(* CoDeSys 2.3.9.41 project: Projmodliv.pro *)
(* Libraries: STANDARD.LIB 4.10.05 10:14:46, IECSFC.LIB 13.4.06 14:51:28, SYSLIBTIME.LIB 12.2.21 12:34:31, SYSTASKINFO.LIB 20.2.06 12:31:38, ANALYZATION.LIB 5.10.99 08:05:06, SYSLIBCALLBACK.LIB 20.2.06 12:31:08, ComService.lib 12.2.21 12:39:42, SysLibCom.lib 12.2.21 12:35:47, ModBus.lib 12.2.21 12:36:21, Util.lib 18.5.10 14:14:28 *)

(* PLC configuration (modules and I/O channels)
DI1 AT %IB0.0 [ByteInput] 8 discrete inputs
Discrete output - relay [ID102] node 1, in %IB1 out %QB1 {PinCount = 1; SafeValueBool = FALSE; Visibility = No}
  DO1 AT %QX1.0 [BitOutput] relay
Discrete output - relay [ID102] node 2, in %IB2 out %QB2 {PinCount = 1; SafeValueBool = FALSE; Visibility = No}
  AT %QX2.0 [BitOutput] relay
Discrete output - relay [ID102] node 3, in %IB3 out %QB3 {PinCount = 1; SafeValueBool = FALSE; Visibility = No}
  AT %QX3.0 [BitOutput] relay
Discrete output - relay [ID102] node 4, in %IB4 out %QB4 {PinCount = 1; SafeValueBool = FALSE; Visibility = No}
  AT %QX4.0 [BitOutput] relay
Discrete output - relay [ID102] node 5, in %IB5 out %QB5 {PinCount = 1; SafeValueBool = FALSE; Visibility = No}
  AT %QX5.0 [BitOutput] relay
  DO6 AT %QX6.0 [BitOutput] relay
AT %QX7.0 [BitOutput] Special output
AT %IW8.0 [WordInput] Cycle time in 100 mks
AT %IW8.1 [WordInput] Time to backup power down, s
AT %ID8.2 [FloatInput] Temp inside PLC
AT %IX8.3 [BitInput] Power status
AT %IX8.4 [BitInput] CPU is overloaded, optimize your programm or increase PLC cycle
AT %IW8.5 [WordInput] Free processor resourse mks in 1 cycle
RS-232 [COM2_USART] node 0, in %IB9.0.0 out %QB9.0.0 {CommunicationSpeed = 9600; Parity = NO PARITY CHECK; BitLength = 8 bits; StopLength = One stop bit; InterfaceType = RS232; FrameOriented = RTU; Timeout = 0; Visibility = No}
ReSlave0 AT %QW9.1.0 [WordOutput]
ReSlave1 AT %QW9.2.0 [WordOutput]
ReSlave2 AT %QW9.3.0 [WordOutput]
ReSlave3 AT %QW9.4.0 [WordOutput]
ReSlave4 AT %QW9.5.0 [WordOutput]
ReSlave5 AT %QW9.6.0 [WordOutput]
ReSlave6 AT %QW9.7.0 [WordOutput]
ReSlave7 AT %QW9.8.0 [WordOutput]
ReSlave8 AT %QW9.9.0 [WordOutput]
ReSlave9 AT %QW9.10.0 [WordOutput]
ReSlave10 AT %QW9.11.0 [WordOutput]
ReSlave11 AT %QW9.12.0 [WordOutput]
ReSlave12 AT %QW9.13.0 [WordOutput]
ReSlave13 AT %QW9.14.0 [WordOutput]
ReSlave14 AT %QW9.15.0 [WordOutput]
ReSlave15 AT %QW9.16.0 [WordOutput]
ReSlave16 AT %QW9.17.0 [WordOutput]
ReSlave17 AT %QW9.18.0 [WordOutput]
ReSlave18 AT %QW9.19.0 [WordOutput]
ReSlave19 AT %QW9.20.0 [WordOutput]
ReSlave20 AT %QW9.21.0 [WordOutput]
ReSlave21 AT %QW9.22.0 [WordOutput]
ReSlave22 AT %QW9.23.0 [WordOutput]
ReSlave23 AT %QW9.24.0 [WordOutput]
ReSlave24 AT %QW9.25.0 [WordOutput]
ReSlave25 AT %QW9.26.0 [WordOutput]
ReSlave26 AT %QW9.27.0 [WordOutput]
ReSlave27 AT %QW9.28.0 [WordOutput]
ReSlave28 AT %QW9.29.0 [WordOutput]
ReSlave29 AT %QW9.30.0 [WordOutput]
ReSlave30 AT %QW9.31.0 [WordOutput]
ReSlave31 AT %QW9.32.0 [WordOutput]
ReSlave32 AT %QW9.33.0 [WordOutput]
ReSlave33 AT %QW9.34.0 [WordOutput]
*)

(* Global variable list: Global_Variables *)
VAR_GLOBAL

	port_opened:  BYTE := 0;
	Settings:COMSETTINGS;
      	com_num: PORTS:=0;
	COM_SERVICE1: COM_SERVICE;

	port_opened2:  BYTE := 0;
	Settings2:COMSETTINGS;
      	com_num2: PORTS:=1;
	COM_SERVICE2: COM_SERVICE;


	ModBusWriteMultiReg232: MB_WR_REGS;
	TonConnect232:ARRAY[0..10] OF  TON;
	ToffConnect232:ARRAY[0..10] OF  TOF;
	ConnectionStatus232:ARRAY[0..10] OF  BOOL;
	Buffer232: ARRAY[0..255] OF BYTE;
	Cmpl232: ARRAY[0..10] OF BOOL;
	Err232: ARRAY[0..10] OF BYTE;
       SCADAData:ARRAY[0..70] OF WORD;

	Buffer: ARRAY[0..255] OF BYTE;
	Cmpl: ARRAY[0..30] OF BOOL;
	Err: ARRAY[0..30] OF BYTE;
	i: BYTE;
	j: BYTE;

      TonConnect: ARRAY[0..3] OF TON;
	ToffConnect: ARRAY[0..3] OF TOF;
	ConnectionStatus: ARRAY [0..3] OF BOOL;



	ModBusWriteMultiCoil: ARRAY[0..1] OF MB_WR_COILS;
	ModBusReadHoldReg: ARRAY[0..10] OF MB_RD_HOLD_REGS;
	ModBusWriteMultiReg: ARRAY[0..10] OF MB_WR_REGS;
      NumberSend: BYTE;

	DisplayData:ARRAY[0..100] OF WORD;

       TimeOut: TIME := T#30ms;

       Out1: WORD;
	 In1: WORD;
       In2: WORD;
	PLCtime:ARRAY[0..10] OF WORD;

      BKDU_KTV:  ARRAY [0..1] OF WORD;  (*BKDU_KTV[0], 5*)

       LocalTime: CurTime;
	TimeL: SysTime64;

	CommCycleTime: SysTime64;
	CommCycleTimePrev: SysTime64;

       ServisWork: BOOL;

	Stop: BOOL;
	StopTime: TIME:=T#1S;
	Zashtibovka: BOOL;
	Zash: BOOL;
	ZashTime: TIME := T#10S;
	KTB: BOOL;
	KTBTime: TIME := T#1S;
	DKS: BOOL;
	DKSTime: TIME := T#10S;
	BOP: INT;
	SirVPN: BOOL;
       AvSirVPN: BOOL;
	TK1: INT;
	TK2: INT;
	TK3: INT;
	TK4: INT;
	KTBStopAv: BOOL;
	KTBStopAvKZ: BOOL;
	KTBCurrent: UINT;
	KTBPower: UINT;
       StopSignal: TP;

	KTBRabotaet: BOOL;
	RazgonStop: BOOL;
	RabotaSpeedStop: BOOL;
	PuskKonveera: BOOL;
	KSLsrabotal: BOOL;
	KSLKZ: BOOL;
	PodtvPusk4: BOOL;
	PodtvPusk3: BOOL;
	myTP22: BOOL;
	PodtvPusk1: BOOL;
	PodtvPusk2: BOOL;
	PP1: BOOL;
	PP2: BOOL;
	PP3: BOOL;
	PP4: BOOL;
	SbrosRazgona: BOOL;
	Parol: UINT := 0;
	ParolStep: UINT := 0;
	Parol1: UINT := 0;
	Parol2: UINT := 0;
	Parol3: UINT := 0;
	GlobalAvariaStop: BOOL;
	DistSignal: BOOL;
	P1Signal: BOOL;

       myTP100: TON;




END_VAR

VAR_GLOBAL RETAIN

	GetTime: CurTimeEx;
	TimeAndDate: SystemTimeDate;
	Sys_Time: SysTime64;
	set_time: BOOL;
	set_date: BOOL;
	MM: UINT:=10;
	SS: UINT;
	HH: UINT:=10;
	D: UINT:=10;
	M: UINT:=10;
	YY: UINT:=20;







	xDO6: TIME := T#6s;
	ZashtibovkaTime: TIME := T#5S;
	RazgonTime: TIME:=T#5s;
	AvariaTime: TIME:=T#10s;
	PuskTime: TIME := T#5s;
	KTBSht: UINT := 5;
	TipK1: UINT := 0;
       TipK1P: TIME:=T#0.2s;
	TipK1T: UINT := 0;
       TipK1UP: TIME:=T#1s;
	TipK2: UINT := 0;
       TipK2P: TIME:=T#0.2s;
	TipK2T: UINT := 0;
       TipK2UP: TIME:=T#1s;
       TipK3: UINT := 0;
       TipK3P: TIME:=T#0.2s;
	TipK3T: UINT := 0;
       TipK3UP: TIME:=T#1s;
       TipK4: UINT := 0;
       TipK4P: TIME:=T#0.2s;
	TipK4T: UINT := 0;
       TipK4UP: TIME:=T#1s;
	NomSpeed: UINT := 20;
	TipDat: UINT:=1;
	DiamKDKS: UINT:=123;
	ImpDKS: UINT:=30;
       Rez: UINT:=300;

	xDO6q: TIME := T#6s;
	ZashtibovkaTimeq: TIME := T#5S;
	RazgonTimeq: TIME:=T#5s;
	AvariaTimeq: TIME:=T#10s;
	PuskTimeq: TIME := T#5s;
	KTBShtq: UINT := 5;
	TipK1q: UINT := 0;
	TipK1Pq: TIME:=T#0.2s;
	TipK1Tq: UINT := 0;
       TipK1UPq: TIME:=T#1s;
	TipK2q: UINT := 0;
       TipK2Pq: TIME:=T#0.2s;
	TipK2Tq: UINT := 0;
       TipK2UPq: TIME:=T#1s;
       TipK3q: UINT := 0;
       TipK3Pq: TIME:=T#0.2s;
	TipK3Tq: UINT := 0;
       TipK3UPq: TIME:=T#1s;
       TipK4q: UINT := 0;
       TipK4Pq: TIME:=T#0.2s;
	TipK4Tq: UINT := 0;
       TipK4UPq: TIME:=T#1s;
	NomSpeedq: UINT := 20;
	TipDatq: UINT:=1;
	DiamKDKSq: UINT:=123;
	ImpDKSq: UINT:=30;
       Rezq: UINT:=300;

	xDO6qi: UINT :=60;
	ZashtibovkaTimeqi: UINT := 50;
	RazgonTimeqi: UINT:=50;
	AvariaTimeqi: WORD:=10;
	PuskTimeqi: WORD := 50;
      TipK1Pqi: UINT:=2;
      TipK1UPqi: UINT:=10;
      TipK2Pqi: UINT:=2;
      TipK2UPqi: UINT:=10;
      TipK3Pqi: UINT:=2;
      TipK3UPqi: UINT:=10;
      TipK4Pqi: UINT:=2;
      TipK4UPqi: UINT:=10;


      Reztek:UINT:=300;

	xDO6Po: UINT :=60;
	ZashtibovkaTimePo: UINT := 50;
	RazgonTimePo: UINT:=50;
	AvariaTimePo: WORD:=10;
	PuskTimePo: WORD := 50;
      TipK1PPo: UINT:=2;
      TipK1UPPo: UINT:=10;
      TipK2PPo: UINT:=2;
      TipK2UPPo: UINT:=10;
      TipK3PPo: UINT:=2;
      TipK3UPPo: UINT:=10;
      TipK4PPo: UINT:=2;
      TipK4UPPo: UINT:=10;


	KTB0: UINT;

        Smoke_sensorQ: BOOL:=TRUE;
       Methane_sensorQ:BOOL:=TRUE;
       Guard_sensorQ:BOOL:=TRUE;
       Add_avarQ:BOOL:=TRUE;



       Smoke_sensor: BOOL:=TRUE;
       Methane_sensor:BOOL:=TRUE;
       Guard_sensor:BOOL:=TRUE;
       Add_avar:BOOL:=TRUE;

END_VAR

(* POU PLC_PRG, ST *)
PROGRAM PLC_PRG
VAR
	myTON:TON;
	myR_TRIG:R_TRIG;
	FI1: INT:=0;

	start: BOOL;

	x: UINT;
	external_event: BOOL;

	ProverkaPuska: INT;
	AvariaSbros: INT;
	AvariaBOP: BOOL;
	ForwardSignal: Signal;
	StartForwardSignal: BOOL;
	Dsignal: BOOL;

       WorkModeF: F_TRIG;
	WorkModeT: R_TRIG;
	StopDist: BOOL;
	RabotaDist: BOOL;
	AvariaDist: BOOL;
	PuskKonveeraN: BOOL;
	a: INT;
	RezNastr: BOOL;
	SwitchWorkMode: BOOL;
	TpAvaria: TP;
	AvariaSirena: BOOL;
      TPBOP: TON;
      TRIGBOP: R_TRIG;
       StopTRIG: F_TRIG;
       StopTRIGr: R_TRIG;
       DistTrig1: R_TRIG;
       DistTrig2: R_TRIG;
	Metka: INT;
      Servis : TON;
      Servis2: TON;
      Servis1: R_TRIG;
	bcdT: INT;
	qwerty: BOOL;
	qwertyTP: TON;
	SmokeAv: BOOL;
	MethanAv: BOOL;
	GuardAv: BOOL;
	AddAv: BOOL;
       StopDistTrig: R_TRIG;
END_VAR
LocalTime(SystemTime:=TimeL );							(*	Функция времени	*)
IF start=0 THEN
	Init();						(*	Открытие порта RS-485	*)
	start:=1;
END_IF
Link();


DisplayData[51].13:=TRUE;

DisplayData[51].6:=TRUE;
DisplayData[51].2:=(ConnectionStatus[0]);       (*БВВ*)
DisplayData[51].3:=(ConnectionStatus[1]);       (*БКДУ*)
DisplayData[51].4:=(ConnectionStatus[2]);       (*ЗАШТЫБОВКА*)
(*IF pollCheclPLZ =16#00FE THEN
pollCheclPLZ :=16#00FF;
ELSE	
pollCheclPLZ :=16#00FE;
END_IF*)
IF DisplayData[23].5=FALSE AND In1.0=TRUE THEN
Servis(In:=In1.4, PT:=t#3s);
IF Servis.Q AND In1.4 THEN
Servis2(In:=In1.1, PT:=t#6s);
Servis1(CLK:=Servis2.Q);
IF Servis1.Q AND In1.4 THEN
ServisWork:=TRUE;
AvariaSbros:=0;

IF TipK1<>2 THEN
Out1.0:=TRUE;
END_IF

IF TipK2<>2 THEN
Out1.1:=TRUE;
END_IF

IF TipK3<>2 THEN
Out1.2:=TRUE;
END_IF

IF TipK4<>2 THEN
Out1.3:=TRUE;
END_IF
END_IF
ELSIF DisplayData[23].5=TRUE AND In1.0=FALSE THEN
ServisWork:=FALSE;
END_IF
END_IF

IF  ServisWork=FALSE THEN
DisplayData[51].5:=FALSE;
ELSE
DisplayData[51].5:=TRUE;
END_IF


StopTRIG(CLK:=In1.0);
StopTRIGr(CLK:=DisplayData[23].5=FALSE);
IF StopTRIGr.Q (*AND StopSignal.Q =FALSE*) THEN
Stop:=FALSE;
END_IF

IF DO1=TRUE THEN
DisplayData[24].15:=TRUE;
ELSIF DO1=FALSE THEN
DisplayData[24].15:=FALSE;
END_IF

IF in1.0=FALSE THEN
DisplayData[23].5:=FALSE;
END_IF

IF ((In1.0=FALSE OR StopTRIG.Q) OR ((KTBRabotaet=FALSE) AND AvariaSbros<>1))  AND ServisWork=FALSE  (*OR StopDist=TRUE*) (*OR RazgonStop=TRUE OR RabotaSpeedStop=TRUE OR KTBRabotaet=FALSE  OR KSLsrabotal=TRUE *)(* OR ((KTBRabotaet=FALSE OR (KSLsrabotal=TRUE AND KSLKZ=FALSE)) AND AvariaSbros<>1)*) THEN
StopDist:=FALSE;
PuskKonveera:=FALSE;
Stop:=TRUE;
sirVPN:=FALSE;
	DO1:=FALSE;
	Out1.0:=FALSE;
	Out1.1:=FALSE;
	Out1.2:=FALSE;
	Out1.3:=FALSE;
RazgonStop:=FALSE;
RabotaSpeedStop:=FALSE;
FI1:=0;
AvariaSbros:=0;

PuskKonveera:=FALSE;

AvariaBOP:=FALSE;

AvariaDist:=FALSE;
P1Signal:=FALSE;

PP1:=TRUE;
PP2:=TRUE;
PP3:=TRUE;
PP4:=TRUE;

Zash:=FALSE;

(*DisplayData[23].5:=TRUE;*)

SbrosRazgona:=TRUE;

PuskKonveera:=FALSE;

GlobalAvariaStop:=FALSE;
SwitchWorkMode:=FALSE;
AvariaSirena:=FALSE;


myTP100(In:=FALSE);
(*IF KTBRabotaet=FALSE  OR KSLsrabotal=TRUE THEN
DisplayData[23].2 :=TRUE;
END_IF
IF RazgonStop=TRUE THEN
END_IF
IF RabotaSpeedStop=TRUE THEN
END_IF*)
ELSIF (RazgonStop=TRUE OR RabotaSpeedStop=TRUE OR KTBstopAvKZ=TRUE OR AvariaBOP=TRUE
(*OR PodtvPusk1=FALSE OR PodtvPusk2=FALSE OR Po           dtvPusk3=FALSE OR PodtvPusk4=FALSE*)
OR  PP1=FALSE OR PP2=FALSE OR PP3=FALSE OR PP4=FALSE OR AvariaDist=TRUE
OR RezNastr=TRUE OR SwitchWorkMode=TRUE
 OR  ConnectionStatus[0]=TRUE OR  ConnectionStatus[1]=TRUE OR ConnectionStatus[2]=TRUE OR SmokeAv=TRUE OR MethanAv=TRUE
OR GuardAv=TRUE OR AddAv=TRUE  )
 AND ServisWork=FALSE THEN
GlobalAvariaStop:=TRUE;
PuskKonveera:=FALSE;
DO1:=FALSE;
Out1.0:=FALSE;
Out1.1:=FALSE;
Out1.2:=FALSE;
Out1.3:=FALSE;
FI1:=2;
AvariaSbros:=1;
DisplayData[23].5:=FALSE;
SbrosRazgona:=TRUE;
AvariaDist:=TRUE;
AvariaSirena:=TRUE;

(*ELSIF KTBRabotaet=FALSE  THEN
PuskKonveera:=FALSE;
DO1:=FALSE;
Out1.0:=FALSE;
Out1.1:=FALSE;
Out1.2:=FALSE;
Out1.3:=FALSE;
FI1:=0;
KTB:=TRUE;
ELSIF DI1.0=TRUE  AND DI1.0=FALSE THEN
PuskKonveera:=FALSE;
DO1:=FALSE;
Out1.0:=FALSE;
Out1.1:=FALSE;
Out1.2:=FALSE;
Out1.3:=FALSE;
FI1:=0;
DKS:=TRUE;*)
ELSIF (SmokeAv=FALSE AND MethanAv=FALSE
AND GuardAv=FALSE AND AddAv=FALSE  )
 AND ServisWork=FALSE AND in1.5=TRUE AND KSLsrabotal=TRUE THEN
DisplayData[23].5:=FALSE;
PuskKonveera:=FALSE;
DO1:=FALSE;
Out1.0:=FALSE;
Out1.1:=FALSE;
Out1.2:=FALSE;
Out1.3:=FALSE;
P1Signal:=FALSE;
SbrosRazgona:=TRUE;
Stop:=TRUE;
AvariaSirena:=TRUE;
myTP100(In:=FALSE);
RazgonStop:=FALSE;
RabotaSpeedStop:=FALSE;
FI1:=0;

ELSIF (SmokeAv=FALSE AND MethanAv=FALSE
AND GuardAv=FALSE AND AddAv=FALSE  )
 AND ServisWork=FALSE AND in1.5=TRUE AND Zash=TRUE THEN
DisplayData[23].5:=FALSE;
PuskKonveera:=FALSE;
DO1:=FALSE;
Out1.0:=FALSE;
Out1.1:=FALSE;
Out1.2:=FALSE;
Out1.3:=FALSE;
P1Signal:=FALSE;
SbrosRazgona:=TRUE;
Stop:=TRUE;
AvariaSirena:=TRUE;
myTP100(In:=FALSE);
RazgonStop:=FALSE;
RabotaSpeedStop:=FALSE;
FI1:=0;

ELSIF (SmokeAv=FALSE AND MethanAv=FALSE
AND GuardAv=FALSE AND AddAv=FALSE  )
 AND ServisWork=FALSE AND in1.5=TRUE AND KSLKZ=TRUE THEN
DisplayData[23].5:=FALSE;
PuskKonveera:=FALSE;
DO1:=FALSE;
Out1.0:=FALSE;
Out1.1:=FALSE;
Out1.2:=FALSE;
Out1.3:=FALSE;
P1Signal:=FALSE;
SbrosRazgona:=TRUE;
Stop:=TRUE;
AvariaSirena:=TRUE;
myTP100(In:=FALSE);
RazgonStop:=FALSE;
RabotaSpeedStop:=FALSE;
FI1:=0;

ELSIF In1.0=FALSE OR In1.4=FALSE AND ServisWork=TRUE THEN
ServisWork:=FALSE;
ELSE
DisplayData[23].5:=TRUE;
AvariaSirena:=FALSE;
(*ELSIF (KTBRabotaet=FALSE OR (KSLsrabotal=TRUE AND KSLKZ=FALSE)) AND AvariaSbros<>1  THEN
PuskKonveera:=FALSE;
Stop:=TRUE;
DO1:=FALSE;
Out1.0:=FALSE;
Out1.1:=FALSE;
Out1.2:=FALSE;
Out1.3:=FALSE;*)
END_IF

IF In1.3=TRUE (*AND ServisWork=FALSE*) THEN
RezNastr:=FALSE;

IF Zashtibovka THEN
DisplayData[23].4:=FALSE;
ELSE
DisplayData[23].4:=TRUE;
END_IF

IF KTBRabotaet=FALSE OR KSLsrabotal=TRUE OR KSLKZ=TRUE OR KTBStopAvKZ THEN
DisplayData[23].2 :=FALSE;
ELSE
DisplayData[23].2 :=TRUE;
END_IF

IF RazgonStop=TRUE OR RabotaSpeedStop=TRUE THEN
DisplayData[23].3:=FALSE;
ELSE
DisplayData[23].3:=TRUE;
END_IF

(*DisplayData[23].3:=DI1.0;*)
(*IF (Zash=FALSE OR KTBRabotaet=TRUE OR RazgonStop=FALSE OR RabotaSpeedStop=FALSE OR KSLsrabotal=FALSE) AND AvariaSbros=0 THEN
DisplayData[23].5:=TRUE;
ELSE
DisplayData[23].5:=FALSE;
END_IF*)


IF In1.4=TRUE THEN
SirVPN:=TRUE;
ELSIF In1.4=FALSE THEN
SirVPN:=FALSE;
END_IF

(*IF In1.0=FALSE THEN
SirVPN:=FALSE;
AvariaSirena:=FALSE;
DO6:=FALSE;
AvSirVPN:=FALSE;
END_IF *)
IF In1.2=FALSE THEN
DisplayData[24].4:=TRUE;
DisplayData[24].5:=FALSE;

(*IF FI1=2 THEN
Stop:=TRUE;
DO1:=FALSE;
Out1.0:=FALSE;
Out1.1:=FALSE;
Out1.2:=FALSE;
Out1.3:=FALSE;
END_IF*)


IF In1.1=TRUE AND FI1=0 AND In1.2=FALSE (*AND DI1.0=FALSE*) AND KSLsrabotal=FALSE (*AND KTBRabotaet=FALSE*) AND KTBstopAvKZ=FALSE  AND Zash=FALSE AND In1.0=TRUE AND AvariaSbros=0 THEN
PuskKonveera:=TRUE;
(*DO1:=TRUE;*)
Stop:=FALSE;
FI1:=1;
SbrosRazgona:=FALSE;
ELSIF In1.1=FALSE AND FI1=1  AND In1.2=FALSE (*AND DI1.0=FALSE*) AND  KSLsrabotal=FALSE (*AND KTBRabotaet=FALSE*) AND KTBstopAvKZ=FALSE AND Zash=FALSE AND In1.0=TRUE AND AvariaSbros=0 THEN
PuskKonveera:=TRUE;
(*DO1:=TRUE;*)
Stop:=FALSE;
SbrosRazgona:=FALSE;
ELSIF In1.1=TRUE AND FI1=1 AND In1.2=FALSE (*AND DI1.0=FALSE*) AND KSLsrabotal=FALSE (*AND KTBRabotaet=FALSE*) AND KTBstopAvKZ=FALSE  AND Zash=FALSE AND In1.0=TRUE AND AvariaSbros=0 THEN
PuskKonveera:=TRUE;
(*DO1:=TRUE;*)
Stop:=FALSE;
SbrosRazgona:=FALSE;
END_IF



ELSIF In1.2=TRUE THEN
DisplayData[24].4:=FALSE;
DisplayData[24].5:=TRUE;
TPBOP(IN:=DI1.1=TRUE AND DI1.2=TRUE , PT:=t#1.0s);
TRIGBOP(CLK:=TPBOP.Q);
DistTrig1(CLK:=(DI1.1=TRUE AND DI1.2=FALSE));
DistTrig2(CLK:=(DI1.1=FALSE AND DI1.2=TRUE));
(*IF FI1=1 THEN
DO1:=FALSE;
Out1.0:=FALSE;
Out1.1:=FALSE;
Out1.2:=FALSE;
Out1.3:=FALSE;
Stop:=TRUE;
END_IF*)
IF DI1.1=TRUE AND DI1.2=FALSE THEN
DisplayData[24].1:=FALSE;
DisplayData[24].2:=TRUE;
DisplayData[24].3:=FALSE;
DisplayData[23].1:=FALSE;
DisplayData[24].6:=FALSE;
ELSIF DI1.1=FALSE AND DI1.2=TRUE THEN
DisplayData[24].1:=TRUE;
DisplayData[24].2:=FALSE;
DisplayData[24].3:=FALSE;
DisplayData[23].1:=FALSE;
DisplayData[24].6:=FALSE;
ELSIF DI1.1=TRUE AND DI1.2=TRUE THEN

DisplayData[24].1:=FALSE;
DisplayData[24].2:=FALSE;
DisplayData[24].3:=FALSE;
DisplayData[24].6:=TRUE;
DisplayData[23].1:=FALSE;
ELSIF DI1.1=FALSE AND DI1.2=FALSE THEN

DisplayData[23].1:=TRUE;
DisplayData[24].1:=FALSE;
DisplayData[24].2:=FALSE;
DisplayData[24].3:=TRUE;
DisplayData[24].6:=FALSE;
END_IF

IF DI1.1=TRUE AND DI1.2=FALSE AND DistTrig1.Q  AND AvariaSbros=0 AND In1.0=TRUE (*AND PuskKonveera=FALSE*) AND AvariaDist=FALSE (*AND Metka=0*) THEN
(*PuskKonveera:=TRUE;*)
(*DO1:=TRUE;*)
(*FI1:=2;*)
RabotaDist:=TRUE;
(*DisplayData[24].1:=FALSE;
DisplayData[24].2:=TRUE;
DisplayData[24].3:=FALSE;
DisplayData[23].1:=FALSE;
DisplayData[24].6:=FALSE;*)
(* Metka:=2;*)
ELSIF DI1.1=FALSE AND DI1.2=TRUE AND DistTrig2.Q AND AvariaSbros=0 AND In1.0=TRUE (*AND PuskKonveera=TRUE  AND RabotaDist=FALSE*) AND AvariaDist=FALSE(* AND Metka=1*) THEN
PuskKonveera:=TRUE;
(*DO1:=TRUE;*)
(*FI1:=2;*)
RabotaDist:=FALSE;
(*DisplayData[24].1:=TRUE;
DisplayData[24].2:=FALSE;
DisplayData[24].3:=FALSE;
DisplayData[23].1:=FALSE;
DisplayData[24].6:=FALSE;*)
SbrosRazgona:=FALSE;
(*Metka:=1;*)

(*PuskKonveera:=TRUE;*)
(*DO1:=TRUE;
FI1:=2;*)


ELSIF (TRIGBOP.Q AND In1.0=TRUE AND AvariaDist=FALSE) OR StopTRIG.Q THEN

Metka:=0;
ProverkaPuska:=0;
(*DisplayData[23].1:=FALSE;*)
DO1:=FALSE;
Out1.0:=FALSE;
Out1.1:=FALSE;
Out1.2:=FALSE;
Out1.3:=FALSE;
(*DisplayData[24].1:=FALSE;
DisplayData[24].2:=FALSE;
DisplayData[24].3:=FALSE;
DisplayData[24].6:=TRUE;*)
StopDist:=TRUE;

SbrosRazgona:=TRUE;
PuskKonveera:=FALSE;
DisplayData[63].13:=TRIGBOP.Q;

(*END_IF*)
ELSIF DI1.1=FALSE AND DI1.2=FALSE AND In1.0=TRUE THEN
DO1:=FALSE;
Out1.0:=FALSE;
Out1.1:=FALSE;
Out1.2:=FALSE;
Out1.3:=FALSE;
AvariaBOP:=TRUE;
(*BOP:=1;
FI1:=1;*)
(*DisplayData[23].1:=TRUE;
DisplayData[24].1:=FALSE;
DisplayData[24].2:=FALSE;
DisplayData[24].3:=TRUE;
DisplayData[24].6:=FALSE;*)
END_IF
END_IF

IF In2<=Reztek THEN
Zashtibovka:=TRUE;
(*B392:=TRUE;*)
ELSIF In2>Reztek THEN
Zashtibovka:=FALSE;
(*B392:=FALSE;*)
END_IF

ELSIF In1.3=FALSE THEN

DO1:=FALSE;
Out1.0:=FALSE;
Out1.1:=FALSE;
Out1.2:=FALSE;
Out1.3:=FALSE;
SirVPN:=FALSE;
RezNastr:=TRUE;
END_IF

IF In1.6=TRUE (*AND TipK1T<>1*) THEN
DisplayData[23].9:=TRUE;
DisplayData[23].10:=FALSE;
ELSIF In1.6=FALSE (*AND TipK1T<>1*) THEN
DisplayData[23].9:=FALSE;
DisplayData[23].10:=TRUE;
END_IF
IF In1.7=TRUE (*AND TipK2T <>1*) THEN
DisplayData[23].11:=TRUE;
DisplayData[23].12:=FALSE;
ELSIF In1.7=FALSE (*AND TipK2T<>1*) THEN
DisplayData[23].11:=FALSE;
DisplayData[23].12:=TRUE;
END_IF
IF In1.8=TRUE (*AND TipK3T<>1*) THEN
DisplayData[23].13:=TRUE;
DisplayData[23].14:=FALSE;
ELSIF In1.8=FALSE (*AND TipK3T<>1*) THEN
DisplayData[23].13:=FALSE;
DisplayData[23].14:=TRUE;
END_IF
IF In1.9=TRUE (*AND TipK4T<>1*) THEN
DisplayData[23].15:=TRUE;
DisplayData[24].0:=FALSE;
ELSIF In1.9=FALSE (*AND TipK4T<>1*) THEN
DisplayData[23].15:=FALSE;
DisplayData[24].0:=TRUE;
END_IF
(********************************************************************************************************
IF TipK1=1 AND DO6=TRUE THEN
out1.0:=TRUE;
ELSIF TipK1<>1 AND DO6=FALSE THEN
out1.0:=FALSE;
END_IF

IF TipK2=1 AND DO6=TRUE THEN
out1.1:=TRUE;
ELSIF TipK2<>1  AND DO6=FALSE THEN
out1.1:=FALSE;
END_IF

IF TipK3=1 AND DO6=TRUE THEN
out1.2:=TRUE;
ELSIF TipK3<>1 AND DO6=FALSE THEN
out1.2:=FALSE;
END_IF

IF TipK4=1 AND DO6=TRUE THEN
out1.3:=TRUE;
ELSIF TipK4<>1 AND DO6=FALSE THEN
out1.3:=FALSE;
END_IF
 ***********************************************************************************************************************)
IF out1.0=TRUE THEN
DisplayData[24].10:=TRUE;
ELSIF out1.0=FALSE THEN
DisplayData[24].10:=FALSE;
END_IF

IF out1.1=TRUE THEN
DisplayData[24].11:=TRUE;
ELSIF out1.1=FALSE THEN
DisplayData[24].11:=FALSE;
END_IF
IF out1.2=TRUE THEN
DisplayData[24].12:=TRUE;
ELSIF out1.2=FALSE THEN
DisplayData[24].12:=FALSE;
END_IF

IF out1.3=TRUE THEN
DisplayData[24].13:=TRUE;
ELSIF out1.3=FALSE THEN
DisplayData[24].13:=FALSE;
END_IF


IF DO6=TRUE THEN
(*Sirena1:='ВКЛ';*)
DisplayData[23].7:=TRUE;
DisplayData[23].8:=FALSE;
ELSIF DO6=FALSE THEN
(*Sirena1:='ВЫКЛ';*)
DisplayData[23].7:=FALSE;
DisplayData[23].8:=TRUE;
END_IF



(**)
IF Smoke_sensor THEN
IF in1.10 THEN
DisplayData[66].8:=TRUE;
DisplayData[66].9:=FALSE;
ELSE
DisplayData[66].8:=FALSE;
DisplayData[66].9:=TRUE;
END_IF
ELSE
IF in1.10=FALSE THEN
DisplayData[66].8:=TRUE;
DisplayData[66].9:=FALSE;
ELSE
DisplayData[66].8:=FALSE;
DisplayData[66].9:=TRUE;
END_IF
END_IF

IF Methane_sensor THEN
IF in1.14 THEN
DisplayData[66].10:=TRUE;
DisplayData[66].11:=FALSE;
ELSE
DisplayData[66].10:=FALSE;
DisplayData[66].11:=TRUE;
END_IF
ELSE
IF in1.14=FALSE THEN
DisplayData[66].10:=TRUE;
DisplayData[66].11:=FALSE;
ELSE
DisplayData[66].10:=FALSE;
DisplayData[66].11:=TRUE;
END_IF
END_IF

IF Guard_sensor THEN
IF in1.15 THEN
DisplayData[66].12:=TRUE;
DisplayData[66].13:=FALSE;
ELSE
DisplayData[66].12:=FALSE;
DisplayData[66].13:=TRUE;
END_IF
ELSE
IF in1.15=FALSE THEN
DisplayData[66].12:=TRUE;
DisplayData[66].13:=FALSE;
ELSE
DisplayData[66].12:=FALSE;
DisplayData[66].13:=TRUE;
END_IF
END_IF

IF  Add_avar THEN
IF in1.5 THEN
DisplayData[66].14:=TRUE;
DisplayData[66].15:=FALSE;
ELSE
DisplayData[66].14:=FALSE;
DisplayData[66].15:=TRUE;
END_IF
ELSE
IF in1.15=FALSE THEN
DisplayData[66].14:=TRUE;
DisplayData[66].15:=FALSE;
ELSE
DisplayData[66].14:=FALSE;
DisplayData[66].15:=TRUE;
END_IF
END_IF

IF DisplayData[66].9=TRUE THEN
SmokeAv:=TRUE;
DisplayData[67].0:=TRUE;
DisplayData[67].1:=FALSE;
ELSE
SmokeAv:=FALSE;
DisplayData[67].0:=FALSE;
DisplayData[67].1:=TRUE;
END_IF

IF DisplayData[66].11=TRUE THEN
MethanAv:=TRUE;
DisplayData[67].2:=TRUE;
DisplayData[67].3:=FALSE;
ELSE
MethanAv:=FALSE;
DisplayData[67].2:=FALSE;
DisplayData[67].3:=TRUE;
END_IF

IF DisplayData[66].13=TRUE THEN
GuardAv:=TRUE;
DisplayData[67].4:=TRUE;
DisplayData[67].5:=FALSE;
ELSE
GuardAv:=FALSE;
DisplayData[67].4:=FALSE;
DisplayData[67].5:=TRUE;
END_IF

IF DisplayData[66].15=TRUE THEN
AddAv:=TRUE;
DisplayData[67].6:=TRUE;
DisplayData[67].7:=FALSE;
ELSE
AddAv:=FALSE;
DisplayData[67].6:=FALSE;
DisplayData[67].7:=TRUE;
END_IF
(**)

Schet();
Timers();
Impuls();
KTBlog();
PuskLogick();
SlaveRS232();


(*IF TK1=1 THEN
IF ProverkaPuska=1 THEN
END_IF
END_IF*)

(*ForwardSignal(Enable:=StartForwardSignal ,Quantity:=4 ,TimeLow:=T#500ms ,TimeHigh:=T#500ms , TimeHighLast:=T#500ms ,Out=> );
Dsignal:=ForwardSignal.Out;
*)
(*
WorkModeT*) 
WorkModeT(CLK:=In1.2);
IF WorkModeT.Q THEN
SwitchWorkMode:=TRUE;
DisplayData[24].1:=FALSE;
DisplayData[24].2:=FALSE;
DisplayData[24].3:=FALSE;
DisplayData[24].6:=TRUE;
DisplayData[51].1:=TRUE;
END_IF

WorkModeF(CLK:=In1.2);
IF WorkModeF.Q THEN
SwitchWorkMode:=TRUE;
DisplayData[24].1:=FALSE;
DisplayData[24].2:=FALSE;
DisplayData[24].3:=FALSE;
DisplayData[24].6:=FALSE;
DisplayData[51].1:=FALSE;
END_IF

IF DI1.3 AND In1.2 THEN
DistSignal:=TRUE;
ELSIF (DI1.3=FALSE AND In1.2) OR (DI1.3 AND In1.2=FALSE) THEN
DistSignal:=FALSE;
END_IF





TpAvaria(IN:=AvariaSirena , PT:=AvariaTime);
IF TpAvaria.Q THEN

IF RazgonStop=TRUE OR RabotaSpeedStop=TRUE THEN
ForwardSignal(Enable:=TpAvaria.Q ,Quantity:=4 ,TimeLow:=T#500ms ,TimeHigh:=T#500ms , TimeHighLast:=T#500ms ,Out=> );
AvSirVPN:=ForwardSignal.Out;
END_IF
IF Zash=TRUE THEN
ForwardSignal(Enable:=TpAvaria.Q ,Quantity:=3 ,TimeLow:=T#500ms ,TimeHigh:=T#500ms , TimeHighLast:=T#500ms ,Out=> );
AvSirVPN:=ForwardSignal.Out;
END_IF
IF KTBstopAvKZ=TRUE OR KSLKZ=TRUE OR KSLsrabotal OR  SmokeAv=TRUE OR MethanAv=TRUE OR GuardAv=TRUE OR AddAv=TRUE THEN (**)
(*ForwardSignal(Enable:=TpAvaria.Q ,Quantity:=3 ,TimeLow:=T#500ms ,TimeHigh:=T#500ms , TimeHighLast:=T#500ms ,Out=> );*)
AvSirVPN:=TpAvaria.Q;
END_IF
IF AvariaBOP=TRUE THEN
ForwardSignal(Enable:=TpAvaria.Q ,Quantity:=3 ,TimeLow:=T#500ms ,TimeHigh:=T#500ms , TimeHighLast:=T#500ms ,Out=> );
AvSirVPN:=ForwardSignal.Out;
END_IF
IF  PP1=FALSE OR PP2=FALSE OR PP3=FALSE OR PP4=FALSE THEN (**)
(*ForwardSignal(Enable:=TpAvaria.Q ,Quantity:=3 ,TimeLow:=T#500ms ,TimeHigh:=T#500ms , TimeHighLast:=T#500ms ,Out=> );*)
AvSirVPN:=TpAvaria.Q;
END_IF
(*ELSIF TpAvaria.Q=FALSE AND AvariaSbros=0 AND SirVPN=FALSE THEN
DO6:=SirVPN;*)
ELSE
AvSirVPN:=FALSE;
END_IF

DisplayData[64]:=In2;


DisplayData[62].10:=Zash;
DisplayData[62].11:=RazgonStop;
DisplayData[62].12:=RabotaSpeedStop;
DisplayData[62].13:=KTBstopAvKZ;
DisplayData[62].14:=KSLKZ;
DisplayData[62].15:=AvariaBOP;
DisplayData[63].0:=NOT PP1;
DisplayData[63].1:=NOT PP2;
DisplayData[63].2:=NOT PP3;
DisplayData[63].3:=NOT PP4;
DisplayData[63].4:=ConnectionStatus[0];
DisplayData[63].5:=ConnectionStatus[1];
DisplayData[63].6:=ConnectionStatus[2];
DisplayData[63].7:=KSLsrabotal;
DisplayData[63].9:=SmokeAv;
DisplayData[63].10:=MethanAv;
DisplayData[63].11:=GuardAv;
DisplayData[63].12:=AddAv;
END_PROGRAM

(* POU Signal, ST *)
FUNCTION_BLOCK Signal
VAR_INPUT
	Enable: BOOL;
	Quantity:BYTE;
	TimeLow: TIME;
	TimeHigh: TIME;
	TimeHighLast: TIME;
	Beep: BOOL;
END_VAR
VAR_OUTPUT
	Out: BOOL;
END_VAR
VAR
	TimeHihgInternal: TIME;
	Work: BOOL;
	Beepp:BLINK;
	BeepLatchQaun: BOOL;
	BeepQaun: BYTE;
END_VAR
IF (Enable OR  Beep)THEN
	Work:=TRUE;
	IF NOT(Beep) THEN
		Beep:=1;
	END_IF
	IF NOT(Out) THEN
		IF BeepLatchQaun THEN
			BeepLatchQaun:=0;
			BeepQaun:=BeepQaun+1;
		END_IF
	ELSE
		BeepLatchQaun:=1;
	END_IF
	IF BeepQaun=(Quantity-1) THEN
		TimeHihgInternal:=TimeHighLast;
	ELSE
		TimeHihgInternal:=TimeHigh;
	END_IF
	IF BeepQaun=Quantity THEN
		Work:=FALSE;
		Beep:=0;
		BeepQaun:=0;
	END_IF
	Beepp(ENABLE:=Beep, TIMELOW:=TimeLow , TIMEHIGH:=TimeHihgInternal, OUT=>Out );
ELSE
	Work:=FALSE;
	Beep:=0;
	BeepQaun:=0;
	Out:=0;
END_IF
END_FUNCTION_BLOCK

(* POU Init, ST *)
FUNCTION Init : BOOL
VAR_INPUT
END_VAR
VAR
END_VAR
WHILE port_opened=0 DO
	IF port_opened=0 THEN
		Settings.Port:=com_num;
		Settings.dwBaudRate:=57600;
		Settings.byParity:=0;
		Settings.dwTimeout:=0;
		Settings.byStopBits:=0;
		Settings.dwBufferSize:=0;
		Settings.dwScan:=0;
	END_IF
	COM_SERVICE1(Enable:=(port_opened=0) , Settings:=Settings , Task:=OPEN_TSK  );
	IF COM_SERVICE1.ready THEN
		port_opened:=2;
	END_IF
END_WHILE
END_FUNCTION

(* POU Link, ST *)
FUNCTION Link : BOOL
VAR_INPUT
END_VAR
VAR
	z: BYTE;
	a: BOOL;

END_VAR
CASE NumberSend OF
0:
	FOR z:=0 TO 70  BY 1 DO
		Buffer[z*2+1]:=WORD_TO_BYTE(DisplayData[z] AND 16#00FF);
		Buffer[z*2]:=WORD_TO_BYTE(SHR(DisplayData[z], 8));
	END_FOR
	ModBusWriteMultiReg[0](
		Enable:=TRUE ,
		Mode:=MB_RTU ,
		DevAddr:=10 ,
		FirstAddr:=305 ,
		Quantity:=85 ,
		ComHandle:=Settings.Port ,
		TimeOut:=T#100ms ,
		Buffer:=Buffer ,
		Complete=>Cmpl[0] ,
		Exception=>Err[0] ,
		RegCnt=> );
	IF(cmpl[0]=TRUE) THEN
		NumberSend:=1;
	END_IF
1:
	       Buffer[1]:=WORD_TO_BYTE(Out1 AND 16#00FF);
	       Buffer[0]:=WORD_TO_BYTE(SHR(Out1, 8));
	       ModBusWriteMultiReg[1](
		Enable:=TRUE ,
		Mode:=MB_RTU ,
		DevAddr:=2 ,
		FirstAddr:=0 ,
		Quantity:=1 ,
		ComHandle:=Settings.Port ,
		TimeOut:=TimeOut ,
		Buffer:=Buffer ,
			Complete=>Cmpl[1] ,
			Exception=>Err[1] ,
			RegCnt=> );
		IF(cmpl[1]=TRUE) THEN
		NumberSend:=2;
	END_IF
2:
IF DisplayData[51].14 THEN
FOR z:=0 TO 5  BY 1 DO
		Buffer[z*2+1]:=WORD_TO_BYTE(PLCtime[z] AND 16#00FF);
		Buffer[z*2]:=WORD_TO_BYTE(SHR(PLCtime[z], 8));
	END_FOR
	ModBusWriteMultiReg[2](
		Enable:=TRUE ,
		Mode:=MB_RTU ,
		DevAddr:=10 ,
		FirstAddr:=220 ,
		Quantity:=5 ,
		ComHandle:=Settings.Port ,
		TimeOut:=T#10ms ,
		Buffer:=Buffer ,
		Complete=>Cmpl[2] ,
		Exception=>Err[2] ,
		RegCnt=> );
	IF(cmpl[2]=TRUE) THEN
		NumberSend:=3;
	END_IF
ELSE
NumberSend:=3;
END_IF

3:
	ModBusReadHoldReg[0](
		Enable:=TRUE ,
		Mode:=MB_RTU ,
		DevAddr:=2 ,
		FirstAddr:=1 ,
		Quantity:=1 ,
		ComHandle:=Settings.Port  ,
		TimeOut:=TimeOut,
		Buffer:=Buffer ,
		Complete=>Cmpl[3] ,
		Exception=>Err[3] ,
		ByteCnt=> );
	IF(cmpl[3]=TRUE) THEN
		IF (Err[3]=0) THEN
			In1:=SHL(Buffer[0], 8)+Buffer[1];
		END_IF
		(*	Фильтр ошибок связи	*)
		TonConnect[0](IN:=((Err[3])<>0) , PT:=T#5s  , Q=>a , ET=> );
		ToffConnect[0](IN:=a , PT:=T#10s , Q=>ConnectionStatus[0] , ET=> );
		NumberSend:=4;
	END_IF
4:
	ModBusReadHoldReg[1](
		Enable:=TRUE ,
		Mode:=MB_RTU ,
		DevAddr:=5 ,
		FirstAddr:=0 ,
		Quantity:=2 ,
		ComHandle:=Settings.Port  ,
		TimeOut:=TimeOut,
		Buffer:=Buffer ,
		Complete=>Cmpl[4] ,
		Exception=>Err[4] ,
		ByteCnt=> );
	IF(cmpl[4]=TRUE) THEN
		IF (Err[4]=0) THEN
			BKDU_KTV[0]:=SHL(Buffer[0], 8)+Buffer[1];
			BKDU_KTV[1]:=SHL(Buffer[2], 8)+Buffer[3];
		END_IF
		(*	Фильтр ошибок связи	*)
		TonConnect[1](IN:=((Err[4])<>0) , PT:=T#5s  , Q=>a , ET=> );
		ToffConnect[1](IN:=a , PT:=T#10s , Q=>ConnectionStatus[1] , ET=> );
		NumberSend:=5;
	END_IF
5:
	ModBusReadHoldReg[2](
		Enable:=TRUE ,
		Mode:=MB_RTU ,
		DevAddr:=32 ,
		FirstAddr:=40001 ,
		Quantity:=1 ,
		ComHandle:=Settings.Port  ,
		TimeOut:=TimeOut,
		Buffer:=Buffer ,
		Complete=>Cmpl[5] ,
		Exception=>Err[5] ,
		ByteCnt=> );
	IF(cmpl[5]=TRUE) THEN
		IF (Err[5]=0) THEN
			In2:=SHL(Buffer[0], 8)+Buffer[1];
		END_IF
		(*	Фильтр ошибок связи	*)
		TonConnect[2](IN:=((Err[5])<>0) , PT:=T#5s  , Q=>a , ET=> );
		ToffConnect[2](IN:=a , PT:=T#10s , Q=>ConnectionStatus[2] , ET=> );
		NumberSend:=6;
	END_IF
6:
	CommCycleTime.ulHigh:=TimeL.ulHigh-CommCycleTimePrev.ulHigh;
	CommCycleTime.ulLow:=TimeL.ulLow-CommCycleTimePrev.ulLow;
	CommCycleTimePrev:=TimeL;
	FOR z:=0 TO 20  BY 1 DO
		cmpl[z]:=FALSE;
	END_FOR
	NumberSend:=0;
END_CASE
END_FUNCTION

(* POU Schet, ST *)
PROGRAM Schet
VAR
	myTON:TON;
	myR_TRIG:R_TRIG;
	myTON1:TON;
	myR_TRIG1:R_TRIG;
	y: BOOL;
       z: BOOL;
	myTON2: TON;
	myR_TRIG2: R_TRIG;
	x: BOOL;

	myTON3: TON;
	myR_TRIG3: R_TRIG;
	q: BOOL;

	myTON0: TON;
	myR_TRIG0: R_TRIG;
	w: BOOL;
	Razreshenie: BOOL;
	myTON9: TON;
	myR_TRIG9: R_TRIG;
	TablStep: UINT := 0;
	myTON8: TON;
	myR_TRIG8: R_TRIG;
	TipK1PqPusk: BOOL;
	TipK1TqTime: BOOL;
	TipK2PqPusk: BOOL;
	RpinG: UINT:=0;
	CheckRP: BOOL;
	myTON5: TON;
	myR_TRIG5: R_TRIG;
	CheckSi: BOOL;
	myTON10: TON;
	myR_TRIG10: R_TRIG;
	eID: INT := 0;

	R_TRIGa: R_TRIG;
	KTBVvod: BOOL;
	eIDTrig: F_TRIG;
       Cheat: R_TRIG;
	timesettings: BOOL;

	RpinGT: BYTE:=1;
	myTON57: TON;
	myR_TRIG57: R_TRIG;
	myTON67: TON;
	myR_TRIG67: R_TRIG;
	myTON17: TON;
	myR_TRIG17: R_TRIG;
	CheckRPs: BOOL;
	CheckSis: BOOL;
	Vc: BOOL;
	Cv: BOOL;
       AvariaEkran: R_TRIG;
      AvEkran :BOOL;

	F_TRIGa: F_TRIG;
	KTBv: BOOL;
END_VAR

VAR_INPUT
	TipK2TqTime: BOOL;
	TipK3PqPusk: BOOL;
	TipK3TqTime: BOOL;
	TipK4PqPusk: BOOL;
	TipK4TqTime: BOOL;
END_VAR
(*(*eIDTrig(CLK:=(In1.3));
IF eIDTrig.Q OR pollCheclPLZ =16#FF   THEN*)
IF pollCheclPLZ =16#00 THEN
pollCheclPLZ :=16#FF;

ELSIF pollCheclPLZ=16#FF THEN

pollCheclPLZ :=16#00;
END_IF
(*END_IF*)*)
IF In1.3=FALSE THEN


myTON10(IN:=(In1.3=FALSE AND (In1.11 OR In1.12) AND Razreshenie=FALSE AND ParolStep=0)  ,PT:=t#0.2s);
myR_TRIG10(CLK:=myTon10.Q);
IF myR_TRIG10.Q   THEN
IF In1.11 AND In1.12=FALSE AND eID>=0 THEN
eID:=eID-1;
IF eID=-1 THEN
eID:=3;
END_IF
ELSIF In1.11=FALSE AND In1.12 AND eID<=3 THEN
eID:=eID+1;
IF eID=4 THEN
eID:=0;
END_IF
END_IF
END_IF

Cheat(CLK:=In1.13);

myTON0(IN:=(In1.3=FALSE AND In1.13 AND Razreshenie=FALSE AND eID=0) OR ( RpinG=1 (*AND CheckRP=TRUE*)   AND In1.3=FALSE AND In1.13)  ,PT:=t#0.5s);
myR_TRIG0(CLK:=myTon0.Q);
IF myR_TRIG0.Q   THEN
IF ParolStep<=4 THEN
ParolStep:=ParolStep+1;
END_IF
END_IF

IF ParolStep>=1 AND ParolStep<=4 AND myTon0.Q=FALSE THEN

myTON2(IN:=(In1.3=FALSE AND In1.11) AND x,PT:=t#0.2s);
myR_TRIG2(CLK:=myTon2.Q);
IF myR_TRIG2.Q   THEN
IF Parol<=8 AND ParolStep=1 THEN
Parol:=Parol+1;
x:=FALSE;
ELSIF ParolStep=2 AND Parol1<=8 THEN
Parol1:=Parol1+1;
x:=FALSE;
ELSIF ParolStep=3 AND Parol2<=8 THEN
Parol2:=Parol2+1;
x:=FALSE;
ELSIF ParolStep=4 AND Parol3<=8 THEN
Parol3:=Parol3+1;
x:=FALSE;
END_IF
ELSIF  myR_TRIG2.Q=FALSE THEN
x:=TRUE;
END_IF


myTON3(IN:=(In1.3=FALSE AND In1.12) AND q,PT:=t#0.2s);
myR_TRIG3(CLK:=myTon3.Q);
IF myR_TRIG3.Q   THEN
IF Parol>=1 AND ParolStep=1 THEN
Parol:=Parol-1;
q:=FALSE;
ELSIF ParolStep=2 AND Parol1>=1 THEN
Parol1:=Parol1-1;
q:=FALSE;
ELSIF ParolStep=3 AND Parol2>=1 THEN
Parol2:=Parol2-1;
q:=FALSE;
ELSIF ParolStep=4 AND Parol3>=1 THEN
Parol3:=Parol3-1;
q:=FALSE;
END_IF
ELSIF  myR_TRIG3.Q=FALSE THEN
q:=TRUE;
END_IF

END_IF

IF ParolStep=5 THEN
IF Parol=0 AND Parol1=0 AND Parol2=0 AND Parol3=2 THEN
xDO6:=xDO6q;
xDO6Po:=xDO6qi;
ZashtibovkaTime:=ZashtibovkaTimeq;
ZashtibovkaTimePo:=ZashtibovkaTimeqi;
RazgonTime:=RazgonTimeq;
RazgonTimePo:=RazgonTimeqi;
AvariaTime:=AvariaTimeq;
AvariaTimePo:=AvariaTimeqi;
PuskTime:=PuskTimeq;
PuskTimePo:=PuskTimeqi;
KTBSht:=KTBShtq;
TipK1:=TipK1q;
TipK1P:=TipK1Pq;
TipK1PPo:=TipK1Pqi;
TipK1T:=TipK1Tq;
TipK1UP:=TipK1UPq;
TipK1UPPo:=TipK1UPqi;
TipK2:=TipK2q;
TipK2P:=TipK2Pq;
TipK2PPo:=TipK2Pqi;
TipK2T:=TipK2Tq;
TipK2UP:=TipK2UPq;
TipK2UPPo:=TipK2UPqi;
TipK3:=TipK3q;
TipK3P:=TipK3Pq;
TipK3PPo:=TipK3Pqi;
TipK3T:=TipK3Tq;
TipK3UP:=TipK3UPq;
TipK3UPPo:=TipK3UPqi;
TipK4:=TipK4q;
TipK4P:=TipK4Pq;
TipK4PPo:=TipK4Pqi;
TipK4T:=TipK4Tq;
TipK4UP:=TipK4UPq;
TipK4UPPo:=TipK4UPqi;
NomSpeed:=NomSpeedq;
TipDat:=TipDatq;
DiamKDKS:=DiamKDKSq;
ImpDKS:=ImpDKSq;
Reztek:=Rezq;
(**)
Smoke_sensor:=Smoke_sensorQ;
Methane_sensor:=Methane_sensorQ;
Guard_sensor:=Guard_sensorQ;
Add_avar:=Add_avarQ;
(**)



(*DisplayData[3]:=DisplayData[25];
DisplayData[4]:=DisplayData[26];
DisplayData[6]:=DisplayData[28];
DisplayData[7]:=DisplayData[29];
DisplayData[8]:=DisplayData[30];
DisplayData[9]:=DisplayData[31];


DisplayData[11]:=DisplayData[33];

DisplayData[12]:=DisplayData[34];

DisplayData[13]:=DisplayData[35];

DisplayData[14]:=DisplayData[36];

DisplayData[15]:=DisplayData[37];

DisplayData[16]:=DisplayData[38];
DisplayData[17]:=DisplayData[39];
DisplayData[18]:=DisplayData[40];
DisplayData[19]:=DisplayData[41];
*)


Razreshenie:=FALSE;
RpinG:=0;
Parol:=0;
Parol1:=0;
Parol2:=0;
Parol3:=0;
ParolStep:=0;
ELSIF Parol=0 AND Parol1=0 AND Parol2=0 AND Parol3=1 THEN
Razreshenie:=TRUE;
RpinG:=1;
Parol:=0;
Parol1:=0;
Parol2:=0;
Parol3:=0;
ParolStep:=0;

ELSIF Parol=1 AND Parol1=1 AND Parol2=0 AND Parol3=0 THEN

timesettings:=TRUE;

Parol:=0;
Parol1:=0;
Parol2:=0;
Parol3:=0;
ParolStep:=0;


ELSIF Parol=0 AND Parol1=0 AND Parol2=0 AND Parol3=9 THEN
Razreshenie:=FALSE;
xDO6:=T#6s;
xDO6q:=T#6s;
xDO6qi:=60;
xDO6Po:=60;
DisplayData[3]:=60;
ZashtibovkaTime:=T#5s;
ZashtibovkaTimeq:=t#5s;
ZashtibovkaTimeqi:=50;
ZashtibovkaTimePo:=50;
DisplayData[4]:=50;
RazgonTime:=T#5s;
RazgonTimeq:=T#5s;
RazgonTimeqi:=50;
RazgonTimePo:=50;
DisplayData[5]:=50;
AvariaTime:=T#10s;
AvariaTimeq:=t#10s;
AvariaTimeqi:=10;
AvariaTimePo:=10;
DisplayData[6]:=10;
PuskTime:=T#5s;
PuskTimeq:=t#5s;
PuskTimeqi:=50;
PuskTimePo:=50;
DisplayData[7]:=450;
KTBSht:=5;
KTBShtq:=5;
DisplayData[8]:=5;
TipK1:=0;
TipK1q:=0;
TipK1P:=T#0.2s;
TipK1Pq:=t#0.2s;
TipK1Pqi:=2;
DisplayData[9]:=2;
TipK1T:=0;
TipK1Tq:=0;
TipK1UP:=T#1s;
TipK1UPq:=t#1s;
TipK1UPqi:=10;
DisplayData[10]:=10;
TipK2:=0;
TipK2q:=0;
TipK2P:=T#0.2s;
TipK2Pq:=T#0.2s;
TipK2Pqi:=2;
DisplayData[11]:=2;
TipK2T:=0;
TipK2Tq:=0;
TipK2UP:=T#1s;
TipK2UPq:=T#1s;
TipK2UPqi:=10;
DisplayData[12]:=10;
TipK3:=0;
TipK3q:=0;
TipK3P:=T#0.2s;
TipK3Pq:=T#0.2s;
TipK3Pqi:=2;
DisplayData[13]:=2;
TipK3T:=0;
TipK3Tq:=0;
TipK3UP:=T#1s;
TipK3UPq:=T#1s;
TipK3UPqi:=10;
DisplayData[14]:=10;
TipK4:=0;
TipK4q:=0;
TipK4P:=T#0.2s;
TipK4Pq:=T#0.2s;
TipK4Pqi:=2;
DisplayData[15]:=2;
TipK4T:=0;
TipK4Tq:=0;
TipK4UP:=T#1s;
TipK4UPq:=T#1s;
TipK4UPqi:=10;
DisplayData[16]:=10;
NomSpeed:=20;
NomSpeedq:=20;
TipDat:=1;
TipDatq:=1;
DiamKDKS:=123;
DiamKDKSq:=123;
ImpDKS:=30;
ImpDKSq:=30;

      TipK1PPo:=2;
      TipK1UPPo:=10;
      TipK2PPo:=2;
      TipK2UPPo:=10;
      TipK3PPo:=2;
      TipK3UPPo:=10;
      TipK4PPo:=2;
      TipK4UPPo:=10;
(**)
Smoke_sensorQ:=TRUE;
Methane_sensorQ:=TRUE;
Guard_sensorQ:=TRUE;
Add_avarQ:=TRUE;

Smoke_sensor:=TRUE;
Methane_sensor:=TRUE;
Guard_sensor:=TRUE;
Add_avar:=TRUE;
(**)


RpinG:=0;
Parol:=0;
Parol1:=0;
Parol2:=0;
Parol3:=0;
ParolStep:=0;

ELSIF Parol=9 AND Parol1=8 AND Parol2=7 AND Parol3=6 THEN
F_TRIGa(CLK:=In1.13);
IF F_TRIGa.Q THEN
KTBv:=TRUE;
END_IF
IF KTBv =FALSE THEN
R_TRIGa(CLK:=In1.13);
END_IF
IF  KTBVvod=FALSE THEN
DisplayData[51].7:=TRUE;
R_TRIGa(CLK:=In1.13);
IF R_TRIGa.Q THEN (*IF KTBv=TRUE AND In1.13=TRUE THEN*)
KTB0:=BKDU_KTV[0];
KTBVvod:=TRUE;
END_IF
ELSIF KTBVvod=TRUE THEN
R_TRIGa(CLK:=In1.13);
IF R_TRIGa.Q THEN (*IF KTBv=TRUE AND In1.13=TRUE THEN *)
KTBCurrent:=((BKDU_KTV[0]-KTB0)/KTBSht);
KTBVvod:=FALSE;
KTBv:=FALSE;
DisplayData[51].7:=FALSE;
ParolStep:=0;
Parol:=0;
Parol1:=0;
Parol2:=0;
Parol3:=0;
END_IF
END_IF
ELSE
ParolStep:=0;
Parol:=0;
Parol1:=0;
Parol2:=0;
Parol3:=0;
END_IF
END_IF
DisplayData[25]:=xDO6qi;
DisplayData[26]:=ZashtibovkaTimeqi;
DisplayData[27]:=RazgonTimeqi;
DisplayData[28]:=AvariaTimeqi;
DisplayData[29]:=PuskTimeqi;
DisplayData[30]:=KTBShtq;
DisplayData[31]:=TipK1Pqi;
DisplayData[32]:=TipK1UPqi;
DisplayData[33]:=TipK2Pqi;
DisplayData[34]:=TipK2UPqi;
DisplayData[35]:=TipK3Pqi;
DisplayData[36]:=TipK3UPqi;
DisplayData[37]:=TipK4Pqi;
DisplayData[38]:=TipK4UPqi;
DisplayData[39]:=NomSpeedq;
DisplayData[40]:=DiamKDKSq;
DisplayData[41]:=ImpDKSq;
DisplayData[0]:=Rezq;
DisplayData[1]:=Reztek;
(**)
IF Smoke_sensorQ THEN
DisplayData[65].0:=TRUE;
DisplayData[65].1:=FALSE;
ELSE
DisplayData[65].0:=FALSE;
DisplayData[65].1:=TRUE;
END_IF

IF Methane_sensorQ THEN
DisplayData[65].2:=TRUE;
DisplayData[65].3:=FALSE;
ELSE
DisplayData[65].2:=FALSE;
DisplayData[65].3:=TRUE;
END_IF

IF Guard_sensorQ THEN
DisplayData[65].4:=TRUE;
DisplayData[65].5:=FALSE;
ELSE
DisplayData[65].4:=FALSE;
DisplayData[65].5:=TRUE;
END_IF

IF Add_avarQ THEN
DisplayData[65].6:=TRUE;
DisplayData[65].7:=FALSE;
ELSE
DisplayData[65].6:=FALSE;
DisplayData[65].7:=TRUE;
END_IF

IF Smoke_sensor THEN
DisplayData[65].8:=TRUE;
DisplayData[65].9:=FALSE;
ELSE
DisplayData[65].8:=FALSE;
DisplayData[65].9:=TRUE;
END_IF

IF Methane_sensor THEN
DisplayData[65].10:=TRUE;
DisplayData[65].11:=FALSE;
ELSE
DisplayData[65].10:=FALSE;
DisplayData[65].11:=TRUE;
END_IF

IF Guard_sensor THEN
DisplayData[65].12:=TRUE;
DisplayData[65].13:=FALSE;
ELSE
DisplayData[65].12:=FALSE;
DisplayData[65].13:=TRUE;
END_IF

IF Add_avar THEN
DisplayData[65].14:=TRUE;
DisplayData[65].15:=FALSE;
ELSE
DisplayData[65].14:=FALSE;
DisplayData[65].15:=TRUE;
END_IF

(**)


IF TipK1q=0 THEN
DisplayData[48].4:=TRUE;
DisplayData[48].5:=FALSE;
DisplayData[48].6:=FALSE;
ELSIF TipK1q=1 THEN
DisplayData[48].4:=FALSE;
DisplayData[48].5:=TRUE;
DisplayData[48].6:=FALSE;
ELSIF TipK1q=2 THEN
DisplayData[48].4:=FALSE;
DisplayData[48].5:=FALSE;
DisplayData[48].6:=TRUE;
END_IF

IF TipK2q=0 THEN
DisplayData[48].7:=TRUE;
DisplayData[48].8:=FALSE;
DisplayData[48].9:=FALSE;
ELSIF TipK2q=1 THEN
DisplayData[48].7:=FALSE;
DisplayData[48].8:=TRUE;
DisplayData[48].9:=FALSE;
ELSIF TipK2q=2 THEN
DisplayData[48].7:=FALSE;
DisplayData[48].8:=FALSE;
DisplayData[48].9:=TRUE;
END_IF

IF TipK3q=0 THEN
DisplayData[48].10:=TRUE;
DisplayData[48].11:=FALSE;
DisplayData[48].12:=FALSE;
ELSIF TipK3q=1 THEN
DisplayData[48].10:=FALSE;
DisplayData[48].11:=TRUE;
DisplayData[48].12:=FALSE;
ELSIF TipK3q=2 THEN
DisplayData[48].10:=FALSE;
DisplayData[48].11:=FALSE;
DisplayData[48].12:=TRUE;
END_IF

IF TipK4q=0 THEN
DisplayData[48].13:=TRUE;
DisplayData[48].14:=FALSE;
DisplayData[48].15:=FALSE;
ELSIF TipK4q=1 THEN
DisplayData[48].13:=FALSE;
DisplayData[48].14:=TRUE;
DisplayData[48].15:=FALSE;
ELSIF TipK4q=2 THEN
DisplayData[48].13:=FALSE;
DisplayData[48].14:=FALSE;
DisplayData[48].15:=TRUE;
END_IF

IF TipDatq=0 THEN
DisplayData[48].3:=TRUE;
DisplayData[48].2:=FALSE;
ELSIF TipDatq=1 THEN
DisplayData[48].3:=FALSE;
DisplayData[48].2:=TRUE;
END_IF




IF Razreshenie=TRUE THEN




myTON5(IN:=(In1.3=FALSE AND In1.13=TRUE) ,PT:=t#0.5s);
myR_TRIG5(CLK:=myTon5.Q);
IF myR_TRIG5.Q AND CheckSi=FALSE AND RpinG<>1 THEN
CheckRP:=TRUE;
CheckSi:=TRUE;
ELSIF myR_TRIG5.Q AND CheckSi=TRUE (*AND RpinG<>1*)  THEN
CheckRP:=FALSE;
CheckSi:=FALSE;
END_IF

myTON(IN:=(In1.3=FALSE AND In1.11) AND y,PT:=t#0.2s);
myR_TRIG(CLK:=myTon.Q);
IF myR_TRIG.Q   THEN
IF RpinG>=1 AND CheckRP=FALSE AND ParolStep=0   THEN
RpinG:=RpinG-1;
y:=FALSE;
IF Rping=0 THEN
Rping:=32;
END_IF
END_IF

IF xDO6q<=T#29.8s AND RpinG=2 AND CheckRP=TRUE  THEN
xDO6q:=xDO6q+t#0.2s;
xDO6qi:=xDO6qi+2;
y:=FALSE;
END_IF
IF  ZashtibovkaTimeq<=t#8.8s AND RpinG=3 AND CheckRP=TRUE THEN
ZashtibovkaTimeq:=ZashtibovkaTimeq+t#0.2s;
ZashtibovkaTimeqi:=ZashtibovkaTimeqi+2;
y:=FALSE;
END_IF
IF RazgonTimeq<=t#29.8s AND RpinG=4 AND CheckRP=TRUE THEN
RazgonTimeq:=RazgonTimeq+t#0.2s;
RazgonTimeqi:=RazgonTimeqi+2;
y:=FALSE;
END_IF
IF AvariaTimeq<=t#59s AND RpinG=5 AND CheckRP=TRUE THEN
AvariaTimeq:=AvariaTimeq+t#1s;
AvariaTimeqi:=AvariaTimeqi+1;
y:=FALSE;
END_IF
IF PuskTimeq<=t#19.8s AND RpinG=6 AND CheckRP=TRUE THEN
PuskTimeq:=PuskTimeq+T#0.2s;
PuskTimeqi:=PuskTimeqi+2;
y:=FALSE;
END_IF
IF KTBShtq<=29 AND RpinG=7 AND CheckRP=TRUE THEN
KTBShtq:=KTBShtq+1;
y:=FALSE;
END_IF

IF TipK1q<2 AND RpinG=17 AND CheckRP=TRUE THEN
TipK1q:=TipK1q+1;
y:=FALSE;
END_IF
IF TipK1Pq<=t#9.8s AND RpinG=18 AND CheckRP=TRUE THEN
TipK1Pq:=TipK1Pq+t#0.2s;
TipK1Pqi:=TipK1Pqi+2;
y:=FALSE;
END_IF
IF TipK1Tq<1 AND RpinG=19 AND CheckRP=TRUE THEN
TipK1Tq:=TipK1Tq+1;
y:=FALSE;
END_IF
IF TipK1UPq<=t#9.8s AND RpinG=20 AND CheckRP=TRUE THEN
TipK1UPq:=TipK1UPq+t#0.2s;
TipK1UPqi:=TipK1UPqi+2;
y:=FALSE;
END_IF

IF TipK2q<2 AND RpinG=21 AND CheckRP=TRUE THEN
TipK2q:=TipK2q+1;
y:=FALSE;
END_IF
IF TipK2Pq<=t#9.8s AND RpinG=22 AND CheckRP=TRUE THEN
TipK2Pq:=TipK2Pq+t#0.2s;
TipK2Pqi:=TipK2Pqi+2;
y:=FALSE;
END_IF
IF TipK2Tq<1 AND RpinG=23 AND CheckRP=TRUE THEN
TipK2Tq:=TipK2Tq+1;
y:=FALSE;
END_IF
IF TipK2UPq<=t#9.8s AND RpinG=24 AND CheckRP=TRUE THEN
TipK2UPq:=TipK2UPq+t#0.2s;
TipK2UPqi:=TipK2UPqi+2;
y:=FALSE;
END_IF

IF TipK3q<2 AND RpinG=25 AND CheckRP=TRUE THEN
TipK3q:=TipK3q+1;
y:=FALSE;
END_IF
IF TipK3Pq<=t#9.8s AND RpinG=26 AND CheckRP=TRUE THEN
TipK3Pq:=TipK3Pq+t#0.2s;
TipK3Pqi:=TipK3Pqi+2;
y:=FALSE;
END_IF
IF TipK3Tq<1 AND RpinG=27 AND CheckRP=TRUE THEN
TipK3Tq:=TipK3Tq+1;
y:=FALSE;
END_IF
IF TipK3UPq<=t#9.8s AND RpinG=28 AND CheckRP=TRUE THEN
TipK3UPq:=TipK3UPq+t#0.2s;
TipK3UPqi:=TipK3UPqi+2;
y:=FALSE;
END_IF

IF TipK4q<2 AND RpinG=29 AND CheckRP=TRUE THEN
TipK4q:=TipK4q+1;
y:=FALSE;
END_IF
IF TipK4Pq<=t#9.8s AND RpinG=30 AND CheckRP=TRUE THEN
TipK4Pq:=TipK4Pq+t#0.2s;
TipK4Pqi:=TipK4Pqi+2;
y:=FALSE;
END_IF
IF TipK4Tq<1 AND RpinG=31 AND CheckRP=TRUE THEN
TipK4Tq:=TipK4Tq+1;
y:=FALSE;
END_IF
IF TipK4UPq<=t#9.8s AND RpinG=32 AND CheckRP=TRUE THEN
TipK4UPq:=TipK4UPq+t#0.2s;
TipK4UPqi:=TipK4UPqi+2;
y:=FALSE;
END_IF

IF NomSpeedq<=69 AND RpinG=8 AND CheckRP=TRUE THEN
NomSpeedq:=NomSpeedq+1;
y:=FALSE;
END_IF

IF TipDatq<1 AND RpinG=9 AND CheckRP=TRUE THEN
TipDatq:=TipDatq+1;
y:=FALSE;
END_IF

IF DiamKDKSq<=290 AND RpinG=10 AND CheckRP=TRUE THEN
DiamKDKSq:=DiamKDKSq+1;
y:=FALSE;
END_IF

IF ImpDKSq<=99 AND RpinG=11 AND CheckRP=TRUE THEN
ImpDKSq:=ImpDKSq+1;
y:=FALSE;
END_IF

IF Rezq<=1000 AND RpinG=12 AND CheckRP=TRUE THEN
Rezq:=Rezq+10;
y:=FALSE;
END_IF
(**)
IF RpinG=13 AND CheckRP=TRUE THEN
Smoke_sensorQ:=TRUE;
y:=FALSE;
END_IF

IF RpinG=14 AND CheckRP=TRUE THEN
Methane_sensorQ:=TRUE;
y:=FALSE;
END_IF

IF RpinG=15 AND CheckRP=TRUE THEN
Guard_sensorQ:=TRUE;
y:=FALSE;
END_IF

IF RpinG=16 AND CheckRP=TRUE THEN
Add_avarQ:=TRUE;
y:=FALSE;
END_IF

(**)
ELSIF  myR_TRIG.Q=FALSE THEN
y:=TRUE;
END_IF

myTON1(IN:=(In1.3=FALSE AND In1.12) AND z,PT:=t#0.2s);
myR_TRIG1(CLK:=myTon1.Q);
IF myR_TRIG1.Q  THEN

IF RpinG<=32 AND CheckRP=FALSE AND ParolStep=0   THEN
RpinG:=RpinG+1;
z:=FALSE;
IF RpinG=33 THEN
RpinG:=1;
END_IF
END_IF

IF xDO6q>=t#0.4s AND RpinG=2 AND CheckRP=TRUE  THEN
xDO6q:=xDO6q-t#0.2s;
xDO6qi:=xDO6qi-2;
z:=FALSE;
END_IF
IF  ZashtibovkaTimeq>=t#0.4s AND RpinG=3 AND CheckRP=TRUE  THEN
ZashtibovkaTimeq:=ZashtibovkaTimeq-t#0.2s;
ZashtibovkaTimeqi:=ZashtibovkaTimeqi-2;
z:=FALSE;
END_IF
IF RazgonTimeq>=t#0.4s AND RpinG=4 AND CheckRP=TRUE  THEN
RazgonTimeq:=RazgonTimeq-t#0.2s;
RazgonTimeqi:=RazgonTimeqi-2;
z:=FALSE;
END_IF
IF AvariaTimeq>=t#2s AND RpinG=5 AND CheckRP=TRUE  THEN
AvariaTimeq:=AvariaTimeq-t#1s;
AvariaTimeqi:=AvariaTimeqi-1;
z:=FALSE;
END_IF
IF PuskTimeq>=t#0.4s AND RpinG=6 AND CheckRP=TRUE  THEN
PuskTimeq:=PuskTimeq-T#0.2s;
PuskTimeqi:=PuskTimeqi-2;
z:=FALSE;
END_IF
IF KTBShtq>=1 AND RpinG=7 AND CheckRP=TRUE  THEN
KTBShtq:=KTBShtq-1;
z:=FALSE;
END_IF

IF TipK1q>=1 AND RpinG=17 AND CheckRP=TRUE  THEN
TipK1q:=TipK1q-1;
z:=FALSE;
END_IF
IF TipK1Pq>=t#0.4s AND RpinG=18 AND CheckRP=TRUE  THEN
TipK1Pq:=TipK1Pq-t#0.2s;
TipK1Pqi:=TipK1Pqi-2;
z:=FALSE;
END_IF
IF TipK1Tq>0 AND RpinG=19 AND CheckRP=TRUE  THEN
TipK1Tq:=TipK1Tq-1;
z:=FALSE;
END_IF
IF TipK1UPq>=t#0.4s AND RpinG=20 AND CheckRP=TRUE  THEN
TipK1UPq:=TipK1UPq-t#0.2s;
TipK1UPqi:=TipK1UPqi-2;
z:=FALSE;
END_IF

IF TipK2q>=1 AND RpinG=21 AND CheckRP=TRUE  THEN
TipK2q:=TipK2q-1;
z:=FALSE;
END_IF
IF TipK2Pq>=t#0.4s AND RpinG=22 AND CheckRP=TRUE  THEN
TipK2Pq:=TipK2Pq-t#0.2s;
TipK2Pqi:=TipK2Pqi-2;
z:=FALSE;
END_IF
IF TipK2Tq>0 AND RpinG=23 AND CheckRP=TRUE  THEN
TipK2Tq:=TipK2Tq-1;
z:=FALSE;
END_IF
IF TipK2UPq>=t#0.4s AND RpinG=24 AND CheckRP=TRUE  THEN
TipK2UPq:=TipK2UPq-t#0.2s;
TipK2UPqi:=TipK2UPqi-2;
z:=FALSE;
END_IF

IF TipK3q>=1 AND RpinG=25 AND CheckRP=TRUE  THEN
TipK3q:=TipK3q-1;
z:=FALSE;
END_IF
IF TipK3Pq>=t#0.4s AND RpinG=26 AND CheckRP=TRUE  THEN
TipK3Pq:=TipK3Pq-t#0.2s;
TipK3Pqi:=TipK3Pqi-2;
z:=FALSE;
END_IF
IF TipK3Tq>0 AND RpinG=27 AND CheckRP=TRUE  THEN
TipK3Tq:=TipK3Tq-1;
z:=FALSE;
END_IF
IF TipK3UPq>=t#0.4s AND RpinG=28 AND CheckRP=TRUE  THEN
TipK3UPq:=TipK3UPq-t#0.2s;
TipK3UPqi:=TipK3UPqi-2;
z:=FALSE;
END_IF

IF TipK4q>=1 AND RpinG=29 AND CheckRP=TRUE  THEN
TipK4q:=TipK4q-1;
z:=FALSE;
END_IF
IF TipK4Pq>=t#0.4s AND RpinG=30 AND CheckRP=TRUE  THEN
TipK4Pq:=TipK4Pq-t#0.2s;
TipK4Pqi:=TipK4Pqi-2;
z:=FALSE;
END_IF
IF TipK4Tq>0 AND RpinG=31 AND CheckRP=TRUE  THEN
TipK4Tq:=TipK4Tq-1;
z:=FALSE;
END_IF
IF TipK4UPq>=t#0.4s AND RpinG=32 AND CheckRP=TRUE  THEN
TipK4UPq:=TipK4UPq-t#0.2s;
TipK4UPqi:=TipK4UPqi-2;
z:=FALSE;
END_IF

IF NomSpeedq>=1 AND RpinG=8 AND CheckRP=TRUE  THEN
NomSpeedq:=NomSpeedq-1;
z:=FALSE;
END_IF

IF TipDatq>0 AND RpinG=9 AND CheckRP=TRUE  THEN
TipDatq:=TipDatq-1;
z:=FALSE;
END_IF

IF DiamKDKSq>=2 AND RpinG=10 AND CheckRP=TRUE  THEN
DiamKDKSq:=DiamKDKSq-1;
z:=FALSE;
END_IF

IF ImpDKSq>=2 AND RpinG=11 AND CheckRP=TRUE  THEN
ImpDKSq:=ImpDKSq-1;
z:=FALSE;
END_IF

IF Rezq>=2 AND RpinG=12 AND CheckRP=TRUE  THEN
Rezq:=Rezq-10;
z:=FALSE;
END_IF
(**)
IF RpinG=13 AND CheckRP=TRUE THEN
Smoke_sensorQ:=FALSE;
z:=FALSE;
END_IF

IF RpinG=14 AND CheckRP=TRUE THEN
Methane_sensorQ:=FALSE;
z:=FALSE;
END_IF

IF RpinG=15 AND CheckRP=TRUE THEN
Guard_sensorQ:=FALSE;
z:=FALSE;
END_IF

IF RpinG=16 AND CheckRP=TRUE THEN
Add_avarQ:=FALSE;
z:=FALSE;
END_IF


(**)
ELSIF  myR_TRIG1.Q=FALSE THEN
z:=TRUE;
END_IF

END_IF




myTON9(IN:=(In1.3=FALSE AND In1.11) ,PT:=t#0.5s);
myR_TRIG9(CLK:=myTon9.Q);
IF myR_TRIG9.Q   THEN
IF TablStep<=26 THEN
TablStep:=TablStep+1;
END_IF
END_IF

myTON8(IN:=(In1.3=FALSE AND In1.12) ,PT:=t#0.5s);
myR_TRIG8(CLK:=myTon8.Q);
IF myR_TRIG8.Q   THEN
IF TablStep>=1 THEN
TablStep:=TablStep-1;
END_IF
END_IF


IF TipK1=0 THEN
TipK1PqPusk:=TRUE;
ELSIF TipK1=1 THEN
TipK1PqPusk:=FALSE;
ELSIF TipK1=2 THEN
TipK1PqPusk:=FALSE;
END_IF

IF TipK1=0 AND TipK1T=0 THEN
TipK1TqTime:=TRUE;
ELSE
TipK1TqTime:=FALSE;
END_IF


IF TipK2=0 THEN
TipK2PqPusk:=TRUE;
ELSIF TipK2=1 THEN
TipK2PqPusk:=FALSE;
ELSIF TipK2=2 THEN
TipK2PqPusk:=FALSE;
END_IF

IF TipK2=0 AND TipK2T=0 THEN
TipK2TqTime:=TRUE;
ELSE
TipK2TqTime:=FALSE;
END_IF


IF TipK3=0 THEN
TipK3PqPusk:=TRUE;
ELSIF TipK3=1 THEN
TipK3PqPusk:=FALSE;
ELSIF TipK3=2 THEN
TipK3PqPusk:=FALSE;
END_IF

IF TipK3=0 AND TipK3T=0 THEN
TipK3TqTime:=TRUE;
ELSE
TipK3TqTime:=FALSE;
END_IF


IF TipK4=0 THEN
TipK4PqPusk:=TRUE;
ELSIF TipK4=1 THEN
TipK4PqPusk:=FALSE;
ELSIF TipK4=2 THEN
TipK4PqPusk:=FALSE;
END_IF

IF TipK4=0 AND TipK4T=0 THEN
TipK4TqTime:=TRUE;
ELSE
TipK4TqTime:=FALSE;
END_IF



IF RpinG=1 THEN
DisplayData[46].0:=TRUE;
ELSE
DisplayData[46].0:=FALSE;
END_IF
IF RpinG=2 THEN
DisplayData[46].1:=TRUE;
ELSE
DisplayData[46].1:=FALSE;
END_IF
IF RpinG=3 THEN
DisplayData[46].2:=TRUE;
ELSE
DisplayData[46].2:=FALSE;
END_IF
IF RpinG=4 THEN
DisplayData[46].3:=TRUE;
ELSE
DisplayData[46].3:=FALSE;
END_IF
IF RpinG=5 THEN
DisplayData[46].4:=TRUE;
ELSE
DisplayData[46].4:=FALSE;
END_IF
IF RpinG=6 THEN
DisplayData[46].5:=TRUE;
ELSE
DisplayData[46].5:=FALSE;
END_IF
IF RpinG=7 THEN
DisplayData[46].6:=TRUE;
ELSE
DisplayData[46].6:=FALSE;
END_IF
IF RpinG=8 THEN
DisplayData[46].7:=TRUE;
ELSE
DisplayData[46].7:=FALSE;
END_IF
IF RpinG=9 THEN
DisplayData[46].8:=TRUE;
ELSE
DisplayData[46].8:=FALSE;
END_IF
IF RpinG=10 THEN
DisplayData[46].9:=TRUE;
ELSE
DisplayData[46].9:=FALSE;
END_IF
IF RpinG=11 THEN
DisplayData[46].10:=TRUE;
ELSE
DisplayData[46].10:=FALSE;
END_IF
IF RpinG=12 THEN
DisplayData[46].11:=TRUE;
ELSE
DisplayData[46].11:=FALSE;
END_IF
(**)
IF RpinG=13 THEN
DisplayData[66].0:=TRUE;
ELSE
DisplayData[66].0:=FALSE;
END_IF
IF RpinG=14 THEN
DisplayData[66].1:=TRUE;
ELSE
DisplayData[66].1:=FALSE;
END_IF
IF RpinG=15 THEN
DisplayData[66].2:=TRUE;
ELSE
DisplayData[66].2:=FALSE;
END_IF
IF RpinG=16 THEN
DisplayData[66].3:=TRUE;
ELSE
DisplayData[66].3:=FALSE;
END_IF
(**)
IF RpinG=17 THEN
DisplayData[46].12:=TRUE;
ELSE
DisplayData[46].12:=FALSE;
END_IF
IF RpinG=18 THEN
DisplayData[46].13:=TRUE;
ELSE
DisplayData[46].13:=FALSE;
END_IF
IF RpinG=19 THEN
DisplayData[46].14:=TRUE;
ELSE
DisplayData[46].14:=FALSE;
END_IF
IF RpinG=20 THEN
DisplayData[46].15:=TRUE;
ELSE
DisplayData[46].15:=FALSE;
END_IF
IF RpinG=21 THEN
DisplayData[47].0:=TRUE;
ELSE
DisplayData[47].0:=FALSE;
END_IF
IF RpinG=22 THEN
DisplayData[47].1:=TRUE;
ELSE
DisplayData[47].1:=FALSE;
END_IF
IF RpinG=23 THEN
DisplayData[47].2:=TRUE;
ELSE
DisplayData[47].2:=FALSE;
END_IF
IF RpinG=24 THEN
DisplayData[47].3:=TRUE;
ELSE
DisplayData[47].3:=FALSE;
END_IF
IF RpinG=25 THEN
DisplayData[47].4:=TRUE;
ELSE
DisplayData[47].4:=FALSE;
END_IF
IF RpinG=26 THEN
DisplayData[47].5:=TRUE;
ELSE
DisplayData[47].5:=FALSE;
END_IF
IF RpinG=27 THEN
DisplayData[47].6:=TRUE;
ELSE
DisplayData[47].6:=FALSE;
END_IF
IF RpinG=28 THEN
DisplayData[47].7:=TRUE;
ELSE
DisplayData[47].7:=FALSE;
END_IF
IF RpinG=29 THEN
DisplayData[47].8:=TRUE;
ELSE
DisplayData[47].8:=FALSE;
END_IF
IF RpinG=30 THEN
DisplayData[47].9:=TRUE;
ELSE
DisplayData[47].9:=FALSE;
END_IF
IF RpinG=31 THEN
DisplayData[47].10:=TRUE;
ELSE
DisplayData[47].10:=FALSE;
END_IF
IF RpinG=32 THEN
DisplayData[47].11:=TRUE;
ELSE
DisplayData[47].11:=FALSE;
END_IF


(*IF  RpinG=1 AND CheckRP=TRUE THEN
B356:=TRUE;
ELSE
B356:=FALSE;
END_IF
*)
IF  RpinG=2 AND CheckRP=TRUE THEN
DisplayData[49].2:=TRUE;
ELSE
DisplayData[49].2:=FALSE;
END_IF

IF  RpinG=3 AND CheckRP=TRUE THEN
DisplayData[49].3:=TRUE;
ELSE
DisplayData[49].3:=FALSE;
END_IF

IF  RpinG=4 AND CheckRP=TRUE THEN
DisplayData[49].4:=TRUE;
ELSE
DisplayData[49].4:=FALSE;
END_IF

IF  RpinG=5 AND CheckRP=TRUE THEN
DisplayData[49].5:=TRUE;
ELSE
DisplayData[49].5:=FALSE;
END_IF

IF  RpinG=6 AND CheckRP=TRUE THEN
DisplayData[49].6:=TRUE;
ELSE
DisplayData[49].6:=FALSE;
END_IF

IF  RpinG=7 AND CheckRP=TRUE THEN
DisplayData[49].7:=TRUE;
ELSE
DisplayData[49].7:=FALSE;
END_IF

IF  RpinG=8 AND CheckRP=TRUE THEN
DisplayData[49].8:=TRUE;
ELSE
DisplayData[49].8:=FALSE;
END_IF

IF  RpinG=9 AND CheckRP=TRUE THEN
DisplayData[49].9:=TRUE;
ELSE
DisplayData[49].9:=FALSE;
END_IF

IF  RpinG=10 AND CheckRP=TRUE THEN
DisplayData[49].10:=TRUE;
ELSE
DisplayData[49].10:=FALSE;
END_IF

IF  RpinG=11 AND CheckRP=TRUE THEN
DisplayData[49].11:=TRUE;
ELSE
DisplayData[49].11:=FALSE;
END_IF

IF  RpinG=12 AND CheckRP=TRUE THEN
DisplayData[49].12:=TRUE;
ELSE
DisplayData[49].12:=FALSE;
END_IF
(**)
IF  RpinG=13 AND CheckRP=TRUE THEN
DisplayData[66].4:=TRUE;
ELSE
DisplayData[66].4:=FALSE;
END_IF
IF  RpinG=14 AND CheckRP=TRUE THEN
DisplayData[66].5:=TRUE;
ELSE
DisplayData[66].5:=FALSE;
END_IF
IF  RpinG=15 AND CheckRP=TRUE THEN
DisplayData[66].6:=TRUE;
ELSE
DisplayData[66].6:=FALSE;
END_IF
IF  RpinG=16 AND CheckRP=TRUE THEN
DisplayData[66].7:=TRUE;
ELSE
DisplayData[66].7:=FALSE;
END_IF
(**)
IF  RpinG=17 AND CheckRP=TRUE THEN
DisplayData[49].13:=TRUE;
ELSE
DisplayData[49].13:=FALSE;
END_IF

IF  RpinG=18 AND CheckRP=TRUE THEN
DisplayData[49].14:=TRUE;
ELSE
DisplayData[49].14:=FALSE;
END_IF

IF  RpinG=19 AND CheckRP=TRUE THEN
DisplayData[49].15:=TRUE;
ELSE
DisplayData[49].15:=FALSE;
END_IF

IF  RpinG=20 AND CheckRP=TRUE THEN
DisplayData[50].0:=TRUE;
ELSE
DisplayData[50].0:=FALSE;
END_IF

IF  RpinG=21 AND CheckRP=TRUE THEN
DisplayData[50].1:=TRUE;
ELSE
DisplayData[50].1:=FALSE;
END_IF

IF  RpinG=22 AND CheckRP=TRUE THEN
DisplayData[50].2:=TRUE;
ELSE
DisplayData[50].2:=FALSE;
END_IF

IF  RpinG=23 AND CheckRP=TRUE THEN
DisplayData[50].3:=TRUE;
ELSE
DisplayData[50].3:=FALSE;
END_IF

IF  RpinG=24 AND CheckRP=TRUE THEN
DisplayData[50].4:=TRUE;
ELSE
DisplayData[50].4:=FALSE;
END_IF

IF  RpinG=25 AND CheckRP=TRUE THEN
DisplayData[50].5:=TRUE;
ELSE
DisplayData[50].5:=FALSE;
END_IF

IF  RpinG=26 AND CheckRP=TRUE THEN
DisplayData[50].6:=TRUE;
ELSE
DisplayData[50].6:=FALSE;
END_IF

IF  RpinG=27 AND CheckRP=TRUE THEN
DisplayData[50].7:=TRUE;
ELSE
DisplayData[50].7:=FALSE;
END_IF

IF  RpinG=28 AND CheckRP=TRUE THEN
DisplayData[50].8:=TRUE;
ELSE
DisplayData[50].8:=FALSE;
END_IF

IF  RpinG=29 AND CheckRP=TRUE THEN
DisplayData[50].9:=TRUE;
ELSE
DisplayData[50].9:=FALSE;
END_IF

IF  RpinG=30 AND CheckRP=TRUE THEN
DisplayData[50].10:=TRUE;
ELSE
DisplayData[50].10:=FALSE;
END_IF

IF  RpinG=31 AND CheckRP=TRUE THEN
DisplayData[50].11:=TRUE;
ELSE
DisplayData[50].11:=FALSE;
END_IF

IF  RpinG=32 AND CheckRP=TRUE THEN
DisplayData[50].12:=TRUE;
ELSE
DisplayData[50].12:=FALSE;
END_IF


(*xDO6qi:=(INT_TO_REAL(REAL_TO_INT(xDO6qi*10.0)))/10.0;
ZashtibovkaTimeqi:=(INT_TO_REAL(REAL_TO_INT(ZashtibovkaTimeqi*10.0)))/10.0;
RazgonTimeqi:=(INT_TO_REAL(REAL_TO_INT(RazgonTimeqi*10.0)))/10.0;
(*AvariaTimeqi:=(INT_TO_REAL(REAL_TO_INT(AvariaTimeqi*10.0)))/10.0;
PuskTimeqi:=(INT_TO_REAL(REAL_TO_INT(PuskTimeqi*10.0)))/10.0;*)
TipK1Pqi:=(INT_TO_REAL(REAL_TO_INT(TipK1Pqi*10.0)))/10.0;
TipK1UPqi:=(INT_TO_REAL(REAL_TO_INT(TipK1UPqi*10.0)))/10.0;
TipK2Pqi:=(INT_TO_REAL(REAL_TO_INT(TipK2Pqi*10.0)))/10.0;
TipK2UPqi:=(INT_TO_REAL(REAL_TO_INT(TipK2UPqi*10.0)))/10.0;
TipK3Pqi:=(INT_TO_REAL(REAL_TO_INT(TipK3Pqi*10.0)))/10.0;
TipK3UPqi:=(INT_TO_REAL(REAL_TO_INT(TipK3UPqi*10.0)))/10.0;
TipK4Pqi:=(INT_TO_REAL(REAL_TO_INT(TipK4Pqi*10.0)))/10.0;
TipK4UPqi:=(INT_TO_REAL(REAL_TO_INT(TipK4UPqi*10.0)))/10.0;
NomSpeedq:=(INT_TO_REAL(REAL_TO_INT(NomSpeedq*10.0)))/10.0;
DiamKDKSq:=(INT_TO_REAL(REAL_TO_INT(DiamKDKSq*10.0)))/10.0;
*)

IF TipK1=0 THEN
DisplayData[21].4:=TRUE;
DisplayData[21].5:=FALSE;
DisplayData[21].6:=FALSE;
TK1:=1;
ELSIF TipK1=1 THEN
DisplayData[21].4:=FALSE;
DisplayData[21].5:=TRUE;
DisplayData[21].6:=FALSE;
TK1:=2;
ELSIF TipK1=2 THEN
DisplayData[21].4:=FALSE;
DisplayData[21].5:=FALSE;
DisplayData[21].6:=TRUE;
TK1:=3;
END_IF

IF TipK2=0 THEN
DisplayData[21].7:=TRUE;
DisplayData[21].8:=FALSE;
DisplayData[21].9:=FALSE;
TK2:=1;
ELSIF TipK2=1 THEN
DisplayData[21].7:=FALSE;
DisplayData[21].8:=TRUE;
DisplayData[21].9:=FALSE;
TK2:=2;
ELSIF TipK2=2 THEN
DisplayData[21].7:=FALSE;
DisplayData[21].8:=FALSE;
DisplayData[21].9:=TRUE;
TK2:=3;
END_IF

IF TipK3=0 THEN
DisplayData[21].10:=TRUE;
DisplayData[21].11:=FALSE;
DisplayData[21].12:=FALSE;
TK3:=1;
ELSIF TipK3=1 THEN
DisplayData[21].10:=FALSE;
DisplayData[21].11:=TRUE;
DisplayData[21].12:=FALSE;
TK3:=2;
ELSIF TipK3=2 THEN
DisplayData[21].10:=FALSE;
DisplayData[21].11:=FALSE;
DisplayData[21].12:=TRUE;
TK3:=3;
END_IF

IF TipK4=0 THEN
DisplayData[21].13:=TRUE;
DisplayData[21].14:=FALSE;
DisplayData[21].15:=FALSE;
TK4:=1;
ELSIF TipK4=1 THEN
DisplayData[21].13:=FALSE;
DisplayData[21].14:=TRUE;
DisplayData[21].15:=FALSE;
TK4:=2;
ELSIF TipK4=2 THEN
DisplayData[21].13:=FALSE;
DisplayData[21].14:=FALSE;
DisplayData[21].15:=TRUE;
TK4:=3;
END_IF



IF TipK1Tq=0 THEN
DisplayData[49].0:=TRUE;
DisplayData[49].1:=FALSE;
ELSIF TipK1Tq=1 THEN
DisplayData[49].0:=FALSE;
DisplayData[49].1:=TRUE;
END_IF

IF TipK2Tq=0 THEN
DisplayData[47].12:=TRUE;
DisplayData[47].13:=FALSE;
ELSIF TipK2Tq=1 THEN
DisplayData[47].12:=FALSE;
DisplayData[47].13:=TRUE;
END_IF

IF TipK3Tq=0 THEN
DisplayData[47].14:=TRUE;
DisplayData[47].15:=FALSE;
ELSIF TipK3Tq=1 THEN
DisplayData[47].14:=FALSE;
DisplayData[47].15:=TRUE;
END_IF

IF TipK4Tq=0 THEN
DisplayData[48].0:=TRUE;
DisplayData[48].1:=FALSE;
ELSIF TipK4Tq=1 THEN
DisplayData[48].0:=FALSE;
DisplayData[48].1:=TRUE;
END_IF


IF TipK1T=0 THEN
DisplayData[22].0:=TRUE;
DisplayData[22].1:=FALSE;
ELSIF TipK1T=1 THEN
DisplayData[22].0:=FALSE;
DisplayData[22].1:=TRUE;
END_IF

IF TipK2T=0 THEN
DisplayData[22].2:=TRUE;
DisplayData[22].3:=FALSE;
ELSIF TipK2T=1 THEN
DisplayData[22].2:=FALSE;
DisplayData[22].3:=TRUE;
END_IF

IF TipK3T=0 THEN
DisplayData[22].4:=TRUE;
DisplayData[22].5:=FALSE;
ELSIF TipK3T=1 THEN
DisplayData[22].4:=FALSE;
DisplayData[22].5:=TRUE;
END_IF

IF TipK4T=0 THEN
DisplayData[22].6:=TRUE;
DisplayData[22].7:=FALSE;
ELSIF TipK4T=1 THEN
DisplayData[22].6:=FALSE;
DisplayData[22].7:=TRUE;
END_IF


DisplayData[3]:=xDO6Po;

DisplayData[4]:=ZashtibovkaTimePo;
DisplayData[5]:=RazgonTimePo;
DisplayData[6]:=AvariaTimePo;
DisplayData[7]:=PuskTimePo;
DisplayData[8]:=KTBSht;

DisplayData[9]:=TipK1PPo;

DisplayData[10]:=TipK1UPPo;

DisplayData[11]:=TipK2PPo;

DisplayData[12]:=TipK2UPPo;

DisplayData[13]:=TipK3PPo;

DisplayData[14]:=TipK3UPPo;

DisplayData[15]:=TipK4PPo;

DisplayData[16]:=TipK4UPPo;

DisplayData[17]:=NomSpeed;

DisplayData[18]:=DiamKDKS;
DisplayData[19]:=ImpDKS;

IF TipDat=0 THEN
DisplayData[22].8:=TRUE;
DisplayData[22].9:=FALSE;
ELSIF TipDat=1 THEN
DisplayData[22].8:=FALSE;
DisplayData[22].9:=TRUE;
END_IF





(*DisplayData[3]:=DisplayData[25];
DisplayData[4]:=DisplayData[26];
DisplayData[6]:=DisplayData[28];
DisplayData[7]:=DisplayData[29];
DisplayData[8]:=DisplayData[30];
DisplayData[9]:=DisplayData[31];


DisplayData[11]:=DisplayData[33];

DisplayData[12]:=DisplayData[34];

DisplayData[13]:=DisplayData[35];

DisplayData[14]:=DisplayData[36];

DisplayData[15]:=DisplayData[37];

DisplayData[16]:=DisplayData[38];
DisplayData[17]:=NomSpeed;
DisplayData[18]:=DiamKDKS;
DisplayData[19]:=ImpDKS;*)
ELSIF  In1.3=TRUE THEN
eID:=0;
Razreshenie:=FALSE;
timesettings:=FALSE;
Parol:=0;
Parol1:=0;
Parol2:=0;
Parol3:=0;
ParolStep:=0;
RpinG:=0;
CheckRPs:=FALSE;
CheckSis:=FALSE;
xDO6q:=xDO6;
xDO6qi:=xDO6Po;
ZashtibovkaTimeq:=ZashtibovkaTime;
ZashtibovkaTimeqi:=ZashtibovkaTimePo;
RazgonTimeq:=RazgonTime;
RazgonTimeqi:=RazgonTimePo;
AvariaTimeq:=AvariaTime;
AvariaTimeqi:=AvariaTimePo;
PuskTimeq:=PuskTime;
PuskTimeqi:=PuskTimePo;
KTBShtq:=KTBSht;
TipK1q:=TipK1;
TipK1Pq:=TipK1P;
TipK1Pqi:=TipK1PPo;
TipK1Tq:=TipK1T;
TipK1UPq:=TipK1UP;
TipK1UPqi:=TipK1UPPo;
TipK2q:=TipK2;
TipK2Pq:=TipK2P;
TipK2Pqi:=TipK2PPo;
TipK2Tq:=TipK2T;
TipK2UPq:=TipK2UP;
TipK2UPqi:=TipK2UPPo;
TipK3q:=TipK3;
TipK3Pq:=TipK3P;
TipK3Pqi:=TipK3PPo;
TipK3Tq:=TipK3T;
TipK3UPq:=TipK3UP;
TipK3UPqi:=TipK3UPPo;
TipK4q:=TipK4;
TipK4Pq:=TipK4P;
TipK4Pqi:=TipK4PPo;
TipK4Tq:=TipK4T;
TipK4UPq:=TipK4UP;
TipK4UPqi:=TipK4UPPo;
NomSpeedq:=NomSpeed;
TipDatq:=TipDat;
DiamKDKSq:=DiamKDKS;
ImpDKSq:=ImpDKS;
Rezq:=Reztek;
(**)
Smoke_sensorQ:=Smoke_sensor;
Methane_sensorQ:=Methane_sensor;
Guard_sensorQ:=Guard_sensor;
Add_avarQ:=Add_avar;
(**)


END_IF

DisplayData[42]:=Parol;
DisplayData[43]:=Parol1;
DisplayData[44]:=Parol2;
DisplayData[45]:=Parol3;


IF Parolstep=1 THEN
DisplayData[50].13:=TRUE;
 ELSIF  Parolstep=2 THEN
DisplayData[50].13:=FALSE;
DisplayData[50].14:=TRUE;
 ELSIF  Parolstep=3 THEN
DisplayData[50].14:=FALSE;
DisplayData[50].15:=TRUE;
 ELSIF Parolstep=4  THEN
(*DisplayData[50].11:=TRUE;*)
DisplayData[50].15:=FALSE;
DisplayData[51].0:=TRUE;
ELSIF ParolStep=5 OR ParolStep=0 THEN
DisplayData[50].13:=FALSE;
DisplayData[50].14:=FALSE;
DisplayData[50].15:=FALSE;
DisplayData[51].0:=FALSE;
END_IF

AvariaEkran(CLK:=In1.13);
IF DisplayData[23].6=TRUE AND AvariaEkran.Q THEN
AvEkran:=TRUE;
ELSIF( In1.3 AND AvEkran AND AvariaEkran.Q) OR In1.3=FALSE THEN
AvEkran:=FALSE;
DisplayData[63].8:=FALSE;
END_IF




IF In1.3=TRUE THEN
timesettings:=FALSE;
CheckRPs:=FALSE;
CheckSis:=FALSE;
RpinGT:=0;
IF AvEkran=FALSE THEN
DisplayData[23].6:=TRUE;
DisplayData[21].0:=FALSE;
DisplayData[21].1:=FALSE;
DisplayData[21].2:=FALSE;
DisplayData[21].3:=FALSE;
DisplayData[63].8:=FALSE;
DisplayData[51].14:=FALSE;
ELSE
DisplayData[23].6:=FALSE;
DisplayData[21].0:=FALSE;
DisplayData[21].1:=FALSE;
DisplayData[21].2:=FALSE;
DisplayData[21].3:=FALSE;
DisplayData[63].8:=TRUE;
DisplayData[51].14:=FALSE;
END_IF
(*ELSIF In1.3=FALSE AND Razreshenie=FALSE AND eID=0 THEN
DisplayData[23].6:=FALSE;
E2:=TRUE;
E3:=FALSE;
E4:=FALSE;
E5:=FALSE;*)
ELSIF ((In1.3=FALSE AND RpinG>=11 AND  RpinG<17 AND Razreshenie=TRUE) OR (In1.3=FALSE AND Razreshenie=FALSE AND eID=1)) AND timesettings=FALSE THEN
DisplayData[23].6:=FALSE;
DisplayData[21].0:=FALSE;
DisplayData[21].1:=TRUE;
DisplayData[21].2:=FALSE;
DisplayData[21].3:=FALSE;
DisplayData[51].14:=FALSE;
ELSIF ((In1.3=FALSE AND RpinG<=10 AND Razreshenie=TRUE) OR (In1.3=FALSE AND Razreshenie=FALSE AND eID=0)) AND timesettings=FALSE  THEN
DisplayData[23].6:=FALSE;
DisplayData[21].0:=TRUE;
DisplayData[21].1:=FALSE;
DisplayData[21].2:=FALSE;
DisplayData[21].3:=FALSE;
DisplayData[51].14:=FALSE;
ELSIF ((In1.3=FALSE AND RpinG>=17 AND  RpinG<25 AND Razreshenie=TRUE) OR (In1.3=FALSE AND Razreshenie=FALSE AND eID=2)) AND timesettings=FALSE THEN
DisplayData[23].6:=FALSE;
DisplayData[21].0:=FALSE;
DisplayData[21].1:=FALSE;
DisplayData[21].2:=TRUE;
DisplayData[21].3:=FALSE;
DisplayData[51].14:=FALSE;
(*ELSIF In1.3=FALSE AND RpinG=18 AND Razreshenie=TRUE THEN
DisplayData[23].6:=FALSE;
E2:=FALSE;
E3:=TRUE;
E4:=FALSE;*)
ELSIF((In1.3=FALSE AND RpinG>=25 AND Razreshenie=TRUE) OR (In1.3=FALSE AND Razreshenie=FALSE AND eID=3)) AND timesettings=FALSE THEN
DisplayData[23].6:=FALSE;
DisplayData[21].0:=FALSE;
DisplayData[21].1:=FALSE;
DisplayData[21].2:=FALSE;
DisplayData[21].3:=TRUE;
DisplayData[51].14:=FALSE;
ELSIF timesettings=TRUE THEN
DisplayData[23].6:=FALSE;
DisplayData[21].0:=FALSE;
DisplayData[21].1:=FALSE;
DisplayData[21].2:=FALSE;
DisplayData[21].3:=FALSE;
DisplayData[51].14:=TRUE;
END_IF
IF DisplayData[51].14=TRUE THEN


myTON57(IN:=(In1.3=FALSE AND In1.13=TRUE AND timesettings ) ,PT:=t#0.5s);
myR_TRIG57(CLK:=myTon57.Q);
IF myR_TRIG57.Q AND CheckSis=FALSE  THEN
CheckRPs:=TRUE;
CheckSis:=TRUE;
ELSIF myR_TRIG57.Q AND CheckSis=TRUE (*AND RpinG<>1*)  THEN
CheckRPs:=FALSE;
CheckSis:=FALSE;
PLCtime[0]:=0;
END_IF

myTON67(IN:=(In1.3=FALSE AND In1.11) AND Cv,PT:=t#0.2s);
myR_TRIG67(CLK:=myTon67.Q);
IF myR_TRIG67.Q   THEN
IF RpinGT>1 AND CheckRPs=FALSE    THEN
RpinGT:=RpinGT-1;
Cv:=FALSE;
END_IF



IF YY<=100 AND RpinGT=1 AND CheckRPs=TRUE THEN
YY:=YY+1;
TimeAndDate.Year:=2000+YY;
GetTime (SystemTime:=Sys_Time , TimeDate:= TimeAndDate);
PLCtime[0]:=INT_TO_BCD(YY);
Cv:=FALSE;
END_IF

IF M<=11 AND RpinGT=2 AND CheckRPs=TRUE THEN
M:=M+1;
TimeAndDate.Month:=M;
GetTime (SystemTime:=Sys_Time , TimeDate:= TimeAndDate);
Cv:=FALSE;
PLCtime[0]:=INT_TO_BCD(M);
END_IF

IF D<=30 AND RpinGT=3 AND CheckRPs=TRUE THEN
D:=D+1;
TimeAndDate.Day:=D;
GetTime (SystemTime:=Sys_Time , TimeDate:= TimeAndDate);
PLCtime[0]:=INT_TO_BCD(D);
Cv:=FALSE;
END_IF

IF HH<=22 AND RpinGT=4 AND CheckRPs=TRUE THEN
HH:=HH+1;
TimeAndDate.Hour:=HH;
GetTime (SystemTime:=Sys_Time , TimeDate:= TimeAndDate);
PLCtime[0]:=INT_TO_BCD(HH);
Cv:=FALSE;
END_IF

IF MM<=58 AND RpinGT=5 AND CheckRPs=TRUE THEN
MM:=MM+1;
TimeAndDate.Minute:=MM;
GetTime (SystemTime:=Sys_Time , TimeDate:= TimeAndDate);
PLCtime[0]:=INT_TO_BCD(MM);
Cv:=FALSE;
END_IF


ELSIF  myR_TRIG67.Q=FALSE THEN
Cv:=TRUE;
END_IF

myTON17(IN:=(In1.3=FALSE AND In1.12) AND Vc,PT:=t#0.2s);
myR_TRIG17(CLK:=myTon17.Q);
IF myR_TRIG17.Q  THEN

IF RpinGT<=4 AND CheckRPs=FALSE  THEN
RpinGT:=RpinGT+1;
Vc:=FALSE;
END_IF



IF YY>=20 AND RpinGT=1 AND CheckRPs=TRUE  THEN
YY:=YY-1;
TimeAndDate.Year:=2000+YY;
GetTime (SystemTime:=Sys_Time , TimeDate:= TimeAndDate);
PLCtime[0]:=INT_TO_BCD(YY);
Vc:=FALSE;
END_IF

IF M>=2 AND RpinGT=2 AND CheckRPs=TRUE  THEN
M:=M-1;
TimeAndDate.Month:=M;
GetTime (SystemTime:=Sys_Time , TimeDate:= TimeAndDate);
PLCtime[0]:=INT_TO_BCD(M);
Vc:=FALSE;
END_IF

IF D>=2 AND RpinGT=3 AND CheckRPs=TRUE  THEN
D:=D-1;
TimeAndDate.Day:=D;
GetTime (SystemTime:=Sys_Time , TimeDate:= TimeAndDate);
PLCtime[0]:=INT_TO_BCD(D);
Vc:=FALSE;
END_IF

IF HH>=1 AND RpinGT=4 AND CheckRPs=TRUE  THEN
HH:=HH-1;
TimeAndDate.Hour:=HH;
GetTime (SystemTime:=Sys_Time , TimeDate:= TimeAndDate);
PLCtime[0]:=INT_TO_BCD(HH);
Vc:=FALSE;
END_IF

IF MM>=1 AND RpinGT=5 AND CheckRPs=TRUE  THEN
MM:=MM-1;
TimeAndDate.Minute:=MM;
GetTime (SystemTime:=Sys_Time , TimeDate:= TimeAndDate);
PLCtime[0]:=INT_TO_BCD(MM);
Vc:=FALSE;
END_IF

ELSIF  myR_TRIG17.Q=FALSE THEN
Vc:=TRUE;
END_IF



END_IF


DisplayData[59]:=UINT_TO_WORD(TimeAndDate.Day);
DisplayData[61]:=UINT_TO_WORD(TimeAndDate.Minute);
DisplayData[60]:=UINT_TO_WORD(TimeAndDate.Hour);
DisplayData[57]:=UINT_TO_WORD(TimeAndDate.Year);
DisplayData[58]:=UINT_TO_WORD(TimeAndDate.Month);




DisplayData[52]:=YY;
DisplayData[53]:=M;
DisplayData[54]:=D;
DisplayData[55]:=HH;
DisplayData[56]:=MM;
IF CheckRPs=FALSE THEN
PLCtime[0]:=0;
TimeAndDate.Day:=0;
TimeAndDate.DayOfWeek :=0;
TimeAndDate.dwHighMsec :=0;
TimeAndDate.dwLowMSecs :=0;
TimeAndDate.Milliseconds :=0;
TimeAndDate.Minute :=0;
TimeAndDate.Second :=0;
TimeAndDate.Hour :=0;
TimeAndDate.Year :=0;
TimeAndDate.Month :=0;
END_IF

GetTime (SystemTime:=Sys_Time , TimeDate:= TimeAndDate);




IF RpinGT=1 THEN
DisplayData[62].0:=TRUE;
ELSE
DisplayData[62].0:=FALSE;
END_IF

IF RpinGT=2 THEN
DisplayData[62].1:=TRUE;
ELSE
DisplayData[62].1:=FALSE;
END_IF

IF RpinGT=3 THEN
DisplayData[62].2:=TRUE;
ELSE
DisplayData[62].2:=FALSE;
END_IF

IF RpinGT=4 THEN
DisplayData[62].3:=TRUE;
ELSE
DisplayData[62].3:=FALSE;
END_IF

IF RpinGT=5 THEN
DisplayData[62].4:=TRUE;
ELSE
DisplayData[62].4:=FALSE;
END_IF

IF CheckRPs=TRUE AND  RpinGT=1 THEN
DisplayData[62].5:=TRUE;
PLCtime[1].0:=TRUE;
ELSE
DisplayData[62].5:=FALSE;
PLCtime[1].0:=FALSE;
END_IF

IF CheckRPs=TRUE AND  RpinGT=2 THEN
DisplayData[62].6:=TRUE;
PLCtime[1].1:=TRUE;
ELSE
DisplayData[62].6:=FALSE;
PLCtime[1].1:=FALSE;
END_IF

IF CheckRPs=TRUE AND  RpinGT=3 THEN
DisplayData[62].7:=TRUE;
PLCtime[1].2:=TRUE;
ELSE
DisplayData[62].7:=FALSE;
PLCtime[1].2:=FALSE;
END_IF

IF CheckRPs=TRUE AND  RpinGT=4 THEN
DisplayData[62].8:=TRUE;
PLCtime[1].3:=TRUE;
ELSE
DisplayData[62].8:=FALSE;
PLCtime[1].3:=FALSE;
END_IF

IF CheckRPs=TRUE AND  RpinGT=5 THEN
DisplayData[62].9:=TRUE;
PLCtime[1].4:=TRUE;
ELSE
DisplayData[62].9:=FALSE;
PLCtime[1].4:=FALSE;
END_IF
END_PROGRAM

(* POU Timers, FBD *)
PROGRAM Timers
VAR

	ZashtibovkaS: TON;
	ZashSignal: TP;
	KTBSignal: TP;
	DKSSignal: TP;
	StopSignal1: BOOL;
	ZashSignal1: BOOL;
	DKSSignal1: BOOL;
	KTBSignal1: BOOL;

	A: BOOL;
END_VAR
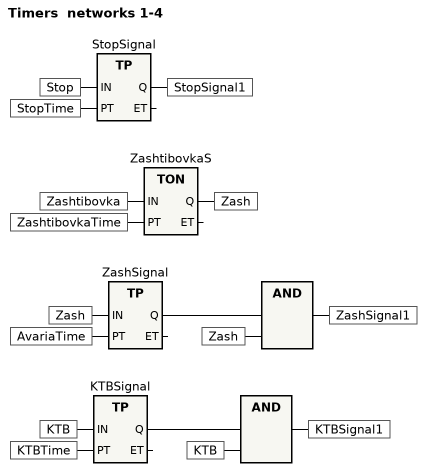
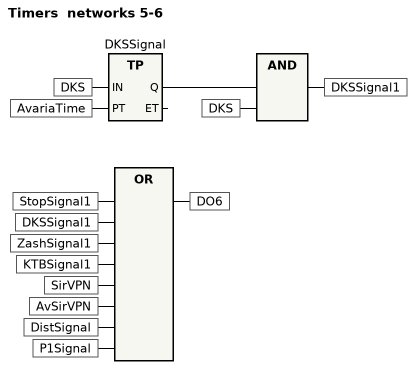
_FBD_ (* Function Block Diagram *)
NETWORK 1
	StopSignal:TP(IN: Stop, PT: StopTime) => StopSignal1
NETWORK 2
	ZashtibovkaS:TON(IN: Zashtibovka, PT: ZashtibovkaTime) => Zash
NETWORK 3
	AND(ZashSignal:TP(IN: Zash, PT: AvariaTime), Zash) => ZashSignal1
NETWORK 4
	AND(KTBSignal:TP(IN: KTB, PT: KTBTime), KTB) => KTBSignal1
NETWORK 5
	AND(DKSSignal:TP(IN: DKS, PT: AvariaTime), DKS) => DKSSignal1
NETWORK 6
	OR(StopSignal1, DKSSignal1, ZashSignal1, KTBSignal1, SirVPN, AvSirVPN, DistSignal, P1Signal) => DO6
_END_FBD_
(* the same logic as Structured Text *)
(* Network 1 *)
StopSignal(IN := Stop, PT := StopTime);
StopSignal1 := StopSignal.Q;
(* Network 2 *)
ZashtibovkaS(IN := Zashtibovka, PT := ZashtibovkaTime);
Zash := ZashtibovkaS.Q;
(* Network 3 *)
ZashSignal(IN := Zash, PT := AvariaTime);
ZashSignal1 := ZashSignal.Q AND Zash;
(* Network 4 *)
KTBSignal(IN := KTB, PT := KTBTime);
KTBSignal1 := KTBSignal.Q AND KTB;
(* Network 5 *)
DKSSignal(IN := DKS, PT := AvariaTime);
DKSSignal1 := DKSSignal.Q AND DKS;
(* Network 6 *)
DO6 := StopSignal1 OR DKSSignal1 OR ZashSignal1 OR KTBSignal1 OR SirVPN OR AvSirVPN OR DistSignal OR P1Signal;
END_PROGRAM

(* POU Impuls, ST *)
PROGRAM Impuls
VAR
	myTON0: TP;
	x: INT;
	myR_TRIG0: R_TRIG;
	y: BOOL:=TRUE;
	C: CTU;
	R_TRIGa: R_TRIG;
	F_TRIGa: F_TRIG;
	sh: INT;
	sh1: INT;

	ss: REAL;
	sl: REAL := 1;
	sm: REAL;
	myTON1: TP;
	q: BOOL:=TRUE;
	w: BOOL;
	R_TRIG2: R_TRIG;

	SpeedTek: REAL;
	SpeedImpulse: REAL;
	RazgonCheck: BOOL;
	myTON2: TP;
	sls: REAL;
	Rdiam: REAL;
	Rimp: REAL;

	myTON3: TON;
	Speedset: BOOL;
	g: REAL;
END_VAR
Rdiam:=UINT_TO_REAL(DiamKDKS);
Rimp:=WORD_TO_REAL(ImpDKS);
Rdiam:=Rdiam/1000;
SpeedImpulse:=((3.1415926535*(Rdiam))/Rimp);
myTON0(IN:=y  ,PT:=t#0.2s);
IF x=1 THEN
y:=TRUE;
END_IF
      IF myTON0.Q =TRUE THEN
R_TRIGa(CLK:=DI1.0);
               IF R_TRIGa.Q THEN
sh:=sh+1;
(*x:=0;*)
                END_IF
x:=0;
       ELSIF myTON0.Q =FALSE AND x=0 THEN
sh1:=sh;
sh:=0;
y:=FALSE;
x:=1;
sl:=sl+0.2;

sl:=(INT_TO_REAL(REAL_TO_INT(sl*10.0)))/10.0;
        END_IF

ss:=sh1*SpeedImpulse*5;
sls:=ss*10;
DisplayData[2]:=REAL_TO_WORD(sls);

g:=(NomSpeed*0.75)/10;

IF (ss<=(NomSpeed*0.75)/10) AND NomSpeed<>0  THEN
Speedset:=TRUE;
ELSIF NomSpeed=0 OR ((ss>(NomSpeed*0.75)/10) AND NomSpeed<>0)  THEN
Speedset:=FALSE;
END_IF
myTON3(IN:=Speedset, PT:=PuskTime);
IF In1.3=TRUE AND ServisWork=FALSE THEN
   IF (Out1.0=TRUE OR Out1.1=TRUE OR  Out1.2=TRUE OR Out1.3=TRUE) AND RazgonTimePo>=3   THEN
myTON1(IN:=(Out1.0 OR Out1.1 OR  Out1.2 OR Out1.3), PT:= RazgonTime);

            IF MyTON1.Q THEN
RazgonCheck:=TRUE;
            ELSE
RazgonCheck:=FALSE;
            END_IF
            IF RazgonCheck=FALSE THEN
                        IF myTON3.Q THEN
RazgonStop:=TRUE;
                        ELSE
RazgonStop:=FALSE;
DO1:=TRUE;
                        END_IF
                        IF RazgonStop=FALSE AND ss<=((NomSpeed*0.75)/10) AND NomSpeed<>0   THEN
(*myTON2(IN:=(ss<=(NomSpeed*0.75) AND  RazgonStop=FALSE ), PT:= PuskTime);*)
                                          IF myTON3.Q AND (ss<=(NomSpeed*0.75)/10) AND RazgonStop=FALSE AND NomSpeed<>0  THEN
RabotaSpeedStop:=TRUE;
                                          ELSE
RabotaSpeedStop:=FALSE;
                                          END_IF
                         END_IF
              END_IF
   ELSIF RazgonTimePo<3 OR SbrosRazgona=TRUE THEN
myTON1(IN:=FALSE);
myTON2(IN:=FALSE);
RazgonCheck:=FALSE;
   END_IF

     IF RazgonStop=TRUE OR RabotaSpeedStop=TRUE THEN
DisplayData[23].0:=TRUE;
     ELSE
DisplayData[23].0:=FALSE;
     END_IF


     IF RazgonCheck=FALSE AND RazgonStop=FALSE AND RazgonTimePo<3  AND (Out1.0=TRUE OR Out1.1=TRUE OR  Out1.2=TRUE OR Out1.3=TRUE)    THEN
DO1:=TRUE;
     ELSIF RazgonCheck=FALSE AND RazgonStop=FALSE AND RazgonTimePo<3 AND (Out1.0=FALSE OR Out1.1=FALSE OR  Out1.2=FALSE OR Out1.3=FALSE) THEN
DO1:=FALSE;
     END_IF

END_IF



(*какого х тут все и без него закрыто но IDE ругается *)
END_PROGRAM

(* POU KTBlog, ST *)
PROGRAM KTBLog
VAR
	KTBOshibka: DINT;
	KTBProsadka: BOOL;
      KTBAvMesto: INT;
END_VAR
IF In1.3=TRUE AND ServisWork=FALSE THEN


IF BKDU_KTV[0]>=32000 THEN
KTBStopAvKZ:=TRUE;
DisplayData[22].10:=TRUE;
ELSE
KTBStopAvKZ:=FALSE;
DisplayData[22].10:=FALSE;
END_IF

KTBPower:=(KTB0+KTBSht*KTBCurrent);
KTBOshibka:=BKDU_KTV[0]-KTB0;
IF KTBPower<=KTBOshibka THEN
KTBProsadka:=TRUE;
ELSE
KTBProsadka:=FALSE;
END_IF

IF BKDU_KTV[0]<=(KTBPower-KTB0) THEN
IF BKDU_KTV[0]<=(KTBCurrent+KTB0+220) AND KTBSht>=1 THEN
KTBAvMesto:=1;
ELSIF  BKDU_KTV[0]<=(2*KTBCurrent+KTB0+220) AND KTBSht>=2 THEN
KTBAvMesto:=2;
ELSIF  BKDU_KTV[0]<=(3*KTBCurrent+KTB0+220) AND KTBSht>=3 THEN
KTBAvMesto:=3;
ELSIF  BKDU_KTV[0]<=(4*KTBCurrent+KTB0+220) AND KTBSht>=4 THEN
KTBAvMesto:=4;
ELSIF  BKDU_KTV[0]<=(5*KTBCurrent+KTB0+220) AND KTBSht>=5 THEN
KTBAvMesto:=5;
ELSIF  BKDU_KTV[0]<=(6*KTBCurrent+KTB0+220) AND KTBSht>=6 THEN
KTBAvMesto:=6;
ELSIF  BKDU_KTV[0]<=(7*KTBCurrent+KTB0+220) AND KTBSht>=7 THEN
KTBAvMesto:=7;
ELSIF  BKDU_KTV[0]<=(8*KTBCurrent+KTB0+220) AND KTBSht>=8 THEN
KTBAvMesto:=8;
ELSIF  BKDU_KTV[0]<=(9*KTBCurrent+KTB0+220) AND KTBSht>=9 THEN
KTBAvMesto:=9;
ELSIF  BKDU_KTV[0]<=(10*KTBCurrent+KTB0+220) AND KTBSht>=10 THEN
KTBAvMesto:=10;
ELSIF  BKDU_KTV[0]<=(11*KTBCurrent+KTB0+220) AND KTBSht>=11 THEN
KTBAvMesto:=11;
ELSIF  BKDU_KTV[0]<=(12*KTBCurrent+KTB0+220) AND KTBSht>=12 THEN
KTBAvMesto:=12;
ELSIF  BKDU_KTV[0]<=(13*KTBCurrent+KTB0+220) AND KTBSht>=13 THEN
KTBAvMesto:=13;
ELSIF  BKDU_KTV[0]<=(14*KTBCurrent+KTB0+220) AND KTBSht>=14 THEN
KTBAvMesto:=14;
ELSIF  BKDU_KTV[0]<=(15*KTBCurrent+KTB0+220) AND KTBSht>=15 THEN
KTBAvMesto:=15;
ELSIF  BKDU_KTV[0]<=(16*KTBCurrent+KTB0+220) AND KTBSht>=16 THEN
KTBAvMesto:=16;
ELSIF  BKDU_KTV[0]<=(17*KTBCurrent+KTB0+220) AND KTBSht>=17 THEN
KTBAvMesto:=17;
ELSIF  BKDU_KTV[0]<=(18*KTBCurrent+KTB0+220) AND KTBSht>=18 THEN
KTBAvMesto:=18;
ELSIF  BKDU_KTV[0]<=(19*KTBCurrent+KTB0+220) AND KTBSht>=19 THEN
KTBAvMesto:=19;
ELSIF  BKDU_KTV[0]<=(20*KTBCurrent+KTB0+220) AND KTBSht>=20 THEN
KTBAvMesto:=20;
ELSIF  BKDU_KTV[0]<=(21*KTBCurrent+KTB0+220) AND KTBSht>=21 THEN
KTBAvMesto:=21;
ELSIF  BKDU_KTV[0]<=(22*KTBCurrent+KTB0+220) AND KTBSht>=22 THEN
KTBAvMesto:=22;
ELSIF  BKDU_KTV[0]<=(23*KTBCurrent+KTB0+220) AND KTBSht>=23 THEN
KTBAvMesto:=23;
ELSIF  BKDU_KTV[0]<=(24*KTBCurrent+KTB0+220) AND KTBSht>=24 THEN
KTBAvMesto:=24;
ELSIF  BKDU_KTV[0]<=(25*KTBCurrent+KTB0+220) AND KTBSht>=25 THEN
KTBAvMesto:=25;
ELSIF  BKDU_KTV[0]<=(26*KTBCurrent+KTB0+220) AND KTBSht>=26 THEN
KTBAvMesto:=26;
ELSIF  BKDU_KTV[0]<=(27*KTBCurrent+KTB0+220) AND KTBSht>=27 THEN
KTBAvMesto:=27;
ELSIF  BKDU_KTV[0]<=(28*KTBCurrent+KTB0+220) AND KTBSht>=28 THEN
KTBAvMesto:=28;
ELSIF  BKDU_KTV[0]<=(29*KTBCurrent+KTB0+220) AND KTBSht>=29 THEN
KTBAvMesto:=29;
ELSIF  BKDU_KTV[0]<=(30*KTBCurrent+KTB0+220) AND KTBSht>=30 THEN
KTBAvMesto:=30;
END_IF
ELSIF BKDU_KTV[0]>(KTBPower-KTB0) THEN
KTBAvMesto:=0;
END_IF
DisplayData[20]:=KTBAvMesto;
IF KTBAvMesto=0 THEN
DisplayData[24].7:=FALSE;
KTBRabotaet:=TRUE;
ELSE
KTBRabotaet:=FALSE;
DisplayData[24].7:=TRUE;
END_IF
(*
KTBRabotaet:=TRUE;
DisplayData[24].7:=FALSE;*)


IF BKDU_KTV[1]=4 OR BKDU_KTV[1]=8 THEN
KSLsrabotal:=FALSE;
KSLKZ:=FALSE;
DisplayData[22].11:=FALSE;
DisplayData[51].12:=FALSE;
ELSIF BKDU_KTV[1]=1 THEN
KSLKZ:=TRUE;
KSLsrabotal:=TRUE;
DisplayData[22].11:=TRUE;
DisplayData[51].12:=FALSE;
ELSIF BKDU_KTV[1]=2 THEN
KSLsrabotal:=TRUE;
KSLKZ:=FALSE;
DisplayData[22].11:=FALSE;
DisplayData[51].12:=TRUE;
END_IF

ELSIF In1.3=TRUE AND ServisWork=TRUE THEN

IF BKDU_KTV[1]=4 OR BKDU_KTV[1]=8 THEN
KSLsrabotal:=FALSE;
KSLKZ:=FALSE;
DisplayData[22].11:=FALSE;
DisplayData[51].12:=FALSE;
ELSIF BKDU_KTV[1]=1 THEN
KSLKZ:=TRUE;
KSLsrabotal:=TRUE;
DisplayData[22].11:=TRUE;
DisplayData[51].12:=FALSE;
ELSIF BKDU_KTV[1]=2 THEN
KSLsrabotal:=TRUE;
KSLKZ:=FALSE;
DisplayData[22].11:=FALSE;
DisplayData[51].12:=TRUE;
END_IF 

END_IF
END_PROGRAM

(* POU PuskLogick, ST *)
PROGRAM PuskLogick
VAR

	SignalMetka: BOOL;
	myTP1: TON;
	myTP10: TON;
	myTP11: TON;
	myTP12: TON;
	myTP13: TON;
	myTP24: TON;
	myTP23: TON;
       myTP22:TON;
	myTP21: TON;

	trig_pusk: R_TRIG;
END_VAR
IF In1.3=TRUE AND ServisWork=FALSE  THEN
(*
IF TipK1T=1 THEN
DisplayData[51].8:=FALSE;
(*DisplayData[23].9:=FALSE;
DisplayData[23].10:=FALSE;*)
ELSE
DisplayData[51].8:=TRUE;
(*DisplayData[23].9:=FALSE;
DisplayData[23].10:=FALSE;*)
END_IF

IF TipK2T=1 THEN
DisplayData[51].9:=FALSE;
(*DisplayData[23].11:=FALSE;
DisplayData[23].12:=FALSE;*)
ELSE
DisplayData[51].9:=TRUE;
(*DisplayData[23].11:=FALSE;
DisplayData[23].12:=FALSE;*)
END_IF

IF TipK3T=1 THEN
DisplayData[51].10:=FALSE;
(*DisplayData[23].13:=FALSE;
DisplayData[23].14:=FALSE;*)
ELSE
DisplayData[51].10:=TRUE;
(*DisplayData[23].13:=FALSE;
DisplayData[23].14:=FALSE;*)
END_IF

IF TipK4T=1 THEN
DisplayData[51].11:=FALSE;
ELSE
DisplayData[51].11:=TRUE;
END_IF
*)


IF TipK1=2 THEN
Out1.0:=FALSE;
DisplayData[22].12:=FALSE;
END_IF

IF TipK2=2 THEN
Out1.1:=FALSE;
DisplayData[22].13:=FALSE;
END_IF

IF TipK3=2 THEN
Out1.2:=FALSE;
DisplayData[22].14:=FALSE;
END_IF

IF TipK4=2 THEN
Out1.3:=FALSE;
DisplayData[22].15:=FALSE;
END_IF


IF PuskKonveera=TRUE AND GlobalAvariaStop=FALSE   THEN
myTP100(IN:=PuskKonveera ,PT:=XDO6);
P1Signal:=NOT(myTP100.Q);
(*P1Signal:=myTP100.Q;*)
IF myTP100.Q=FALSE THEN
SignalMetka:=TRUE;
END_IF
IF SignalMetka THEN
myTP1(IN:=PuskKonveera ,PT:=XDO6);

IF TipK1=1 THEN
Out1.0:=NOT(myTP1.Q);
END_IF

IF TipK2=1 THEN
Out1.1:=NOT(myTP1.Q);
END_IF

IF TipK3=1 THEN
Out1.2:=NOT(myTP1.Q);
END_IF

IF TipK4=1 THEN
Out1.3:=NOT(myTP1.Q); (*Izmenit vezde*)
END_IF

END_IF

ELSIF PuskKonveera=FALSE THEN
myTP100(In:=FALSE);
myTP1(In:=FALSE);
END_IF


IF PuskKonveera=TRUE AND myTP100.Q=TRUE AND SignalMetka=TRUE THEN

IF TipK1=0 THEN
myTP10(IN:=PuskKonveera ,PT:=TipK1P);
IF myTP10.Q=FALSE THEN
Out1.0:=FALSE;
ELSIF myTP10.Q=TRUE THEN
Out1.0:=TRUE;
IF TipK1T=0 THEN
myTP21(IN:=PuskKonveera ,PT:=TipK1UP);
IF myTP21.Q=TRUE AND In1.6=FALSE  THEN
Out1.0:=FALSE;
PodtvPusk1:=FALSE;
PP1:=FALSE;
END_IF
END_IF
END_IF
END_IF

IF TipK2=0 THEN
myTP11(IN:=PuskKonveera ,PT:=TipK2P);
IF myTP11.Q=FALSE THEN
Out1.1:=FALSE;
ELSIF myTP11.Q=TRUE THEN
Out1.1:=TRUE;
IF TipK2T=0 THEN
myTP22(IN:=PuskKonveera ,PT:=TipK2UP);
IF myTP22.Q=TRUE AND In1.7=FALSE  THEN
Out1.1:=FALSE;
PodtvPusk2:=FALSE;
PP2:=FALSE;
END_IF
END_IF
END_IF
END_IF

IF TipK3=0 THEN
myTP12(IN:=PuskKonveera ,PT:=TipK3P);
IF myTP12.Q=FALSE THEN
Out1.2:=FALSE;
ELSIF myTP12.Q=TRUE THEN
Out1.2:=TRUE;
IF TipK3T=0 THEN
myTP23(IN:=PuskKonveera ,PT:=TipK3UP);
IF myTP23.Q=TRUE AND In1.8=FALSE  THEN
Out1.2:=FALSE;
PodtvPusk3:=FALSE;
PP3:=FALSE;
END_IF
END_IF
END_IF
END_IF

IF TipK4=0 THEN
myTP13(IN:=PuskKonveera ,PT:=TipK4P);
IF myTP13.Q=FALSE THEN
Out1.3:=FALSE;
ELSIF myTP13.Q=TRUE THEN
Out1.3:=TRUE;
IF TipK4T=0 THEN
myTP24(IN:=PuskKonveera ,PT:=TipK4UP);
IF myTP24.Q=TRUE AND In1.9=FALSE  THEN
Out1.3:=FALSE;
PodtvPusk4:=FALSE;
PP4:=FALSE;
END_IF
END_IF
END_IF
END_IF

(*END_IF*)

ELSIF PuskKonveera=FALSE THEN
SignalMetka:=FALSE;
myTP100(In:=FALSE);
myTP10(IN:=FALSE);
myTP11(IN:=FALSE);
myTP12(IN:=FALSE);
myTP13(IN:=FALSE);
myTP21(IN:=FALSE);
myTP22(IN:=FALSE);
myTP23(IN:=FALSE);
myTP24(IN:=FALSE);
IF GlobalAvariaStop=TRUE THEN
Out1.0:=FALSE;
Out1.1:=FALSE;
Out1.2:=FALSE;
Out1.3:=FALSE;
myTP100(In:=FALSE);
myTP10(IN:=FALSE);
myTP11(IN:=FALSE);
myTP12(IN:=FALSE);
myTP13(IN:=FALSE);
myTP21(IN:=FALSE);
myTP22(IN:=FALSE);
myTP23(IN:=FALSE);
myTP24(IN:=FALSE);
END_IF
END_IF

IF PP1=FALSE AND  TipK1T=0 AND  PP1=FALSE THEN
(*DisplayData[23].9:=FALSE;
DisplayData[23].10:=TRUE;*)
DisplayData[22].12:=TRUE;
ELSIF (PP1=TRUE AND  TipK1T=0) OR TipK1T=1 THEN
(*DisplayData[23].9:=TRUE;
DisplayData[23].10:=FALSE;*)
DisplayData[22].12:=FALSE;
END_IF

IF PP2=FALSE AND  TipK2T=0 AND  PP2=FALSE THEN
(*DisplayData[23].11:=FALSE;
DisplayData[23].12:=TRUE;*)
DisplayData[22].13:=TRUE;
ELSIF  (PP2=TRUE AND  TipK2T=0)  OR TipK2T=1 THEN
(*DisplayData[23].11:=TRUE;
DisplayData[23].12:=FALSE;*)
DisplayData[22].13:=FALSE;
END_IF

IF PP3=FALSE AND  TipK3T=0 AND  PP3=FALSE THEN
(*DisplayData[23].13:=FALSE;
DisplayData[23].14:=TRUE;*)
DisplayData[22].14:=TRUE;
ELSIF (PP3=TRUE AND  TipK3T=0) OR TipK3T=1 THEN
(*DisplayData[23].13:=TRUE;
DisplayData[23].14:=FALSE;*)
DisplayData[22].14:=FALSE;
END_IF

IF PP4=FALSE AND  TipK4T=0 AND  PP4=FALSE THEN
(*DisplayData[23].15:=FALSE;
DisplayData[24].0:=TRUE;*)
DisplayData[22].15:=TRUE;
ELSIF (PP4=TRUE AND  TipK4T=0) OR TipK4T=1 THEN
(*DisplayData[23].15:=TRUE;
DisplayData[24].0:=FALSE;*)
DisplayData[22].15:=FALSE;
END_IF


END_IF
END_PROGRAM

(* POU SlaveRS232, ST *)
PROGRAM SlaveRS232
VAR
END_VAR
(*IF ReSlave0=1 THEN



IF xDO6>T#30s OR xDO6<T#0.2s  THEN
xDO6:=T#30s;
xDO6Po:=30;

END_IF
IF  ZashtibovkaTime>t#9s OR ZashtibovkaTime<t#0.2s  THEN
ZashtibovkaTime:=t#9s;
ZashtibovkaTimePo:=9;

END_IF
IF RazgonTime>t#10s OR RazgonTime<t#0.2s   THEN
RazgonTime:=t#10s;
RazgonTimePo:=10;

END_IF
IF AvariaTime>t#60s OR AvariaTime<t#1s THEN
AvariaTime:=t#60s;
AvariaTimePo:=60;

END_IF
IF PuskTime>t#20s  OR PuskTime<t#0.2s THEN
PuskTime:=T#20s;
PuskTimePo:=20;
END_IF

IF KTBSht>30  OR KTBSht<30 THEN
KTBSht:=30;
END_IF

IF TipK1>2 OR TipK1<0 THEN
TipK1:=2;

END_IF
IF TipK1P>t#10s OR TipK1P<t#0.2s THEN
TipK1P:=t#10s;
TipK1PPo:=10;

END_IF
IF TipK1T>1 OR TipK1T<0  THEN
TipK1T:=1;

END_IF
IF TipK1UP>t#10s OR TipK1UP<t#0.2s THEN
TipK1UP:=t#10s;
TipK1UPPo:=10;

END_IF

IF TipK2>2 OR TipK2<0  THEN
TipK2:=2;

END_IF
IF TipK2P>t#10s OR TipK2P<t#0.2s THEN
TipK2P:=t#10s;
TipK2PPo:=10;

END_IF
IF TipK2T>1 OR TipK2T<0 THEN
TipK2T:=1;

END_IF
IF TipK2UP>t#10s OR TipK2UP<t#0.2s THEN
TipK2UP:=t#10s;
TipK2UPPo:=10;

END_IF

IF TipK3>2  OR TipK3<0 THEN
TipK3:=2;

END_IF
IF TipK3P>t#10s OR TipK3P<t#0.2s THEN
TipK3P:=t#10s;
TipK3PPo:=10;

END_IF
IF TipK3T>1 OR TipK3T<0  THEN
TipK3T:=1;

END_IF
IF TipK3UP>t#10s OR TipK3UP<t#0.2s  THEN
TipK3UP:=t#10s;
TipK3UPPo:=10;

END_IF

IF TipK4>2 OR TipK4<0  THEN
TipK4:=2;

END_IF
IF TipK4P>t#10s OR TipK4P<t#0.2s  THEN
TipK4P:=t#10s;
TipK4PPo:=10;

END_IF
IF TipK4T>1  OR TipK4T<0  THEN
TipK4T:=1;

END_IF
IF TipK4UP>t#10s OR  TipK4UP<t#0.2s   THEN
TipK4UP:=t#10s;
TipK4UPPo:=10;

END_IF

IF NomSpeed>70 OR NomSpeed<0 THEN
NomSpeed:=70;

END_IF

IF TipDat>1 OR  TipDat<0 THEN
TipDat:=1;

END_IF

IF DiamKDKS>291 OR DiamKDKS<1   THEN
DiamKDKS:=291;

END_IF

IF ImpDKS>100 OR ImpDKS<1  THEN
ImpDKS:=1;

END_IF

IF Rez>1000 OR Rez<0 THEN
Rez:=1000;

END_IF


END_IF*)
ReSlave1:=DisplayData[3]; (*Время звучания сирены при пуске (контакт DO6 ПЛК), с*)
ReSlave2:=DisplayData[4]; (*Время на отключение конвейера при заштыбовке (чувствительность фильтра)*)
ReSlave3:=DisplayData[5]; (*Время разгона конвейера (нечувствительность датчика скорости, 0.2 - ДС игнорируется)*)
ReSlave4:=DisplayData[6]; (*Время звучания сирены при аварии*)
ReSlave5:=DisplayData[7]; (*Время отключения по скорости (<75%)*)
ReSlave6:=DisplayData[8]; (*Количество КТВ*)
ReSlave7:=DisplayData[19]; (*Количество импульсов на оборот датчика ДМ*)
ReSlave8:=TipK1;                    (*Тип контакта *)
ReSlave9:=DisplayData[9];    (*Время включения контакта 1*)
ReSlave10:=TipK1T;                 (*Подтверждение включения пускателя *)
ReSlave11:=DisplayData[10]; (*Время подтверждения включения пускателя *)
ReSlave12:=TipK2;
ReSlave13:=DisplayData[11];
ReSlave14:=TipK2T;
ReSlave15:=DisplayData[12];
ReSlave16:=TipK3;
ReSlave17:=DisplayData[13];
ReSlave18:=TipK3T;
ReSlave19:=DisplayData[14];
ReSlave20:=TipK4;
ReSlave21:=DisplayData[15];
ReSlave22:=TipK4T;
ReSlave23:=DisplayData[16];
ReSlave24:=DisplayData[17]; (*Номинальная скорость конвейера*)
ReSlave25:=DisplayData[18]; (*Диаметр колеса ДМ (см) *)
ReSlave26:=DisplayData[1];    (*Сопротивление при заштыбовке кОМ*)
ReSlave27:=DisplayData[2]; (*Скорость*)
ReSlave28:=TipDat;                (*Тип датчика скорости*)
ReSlave29:=DisplayData[64]; (*Сопротивлние тек*)
(*eSlave30 Аварии*)
ReSlave30.0:=DisplayData[62].10;
ReSlave30.1:=DisplayData[62].11;
ReSlave30.2:=DisplayData[62].12;
ReSlave30.3:=DisplayData[62].13;
ReSlave30.4:=DisplayData[62].14;
ReSlave30.5:=DisplayData[62].15;
ReSlave30.6:=DisplayData[63].0;
ReSlave30.7:=DisplayData[63].1;
ReSlave30.8:=DisplayData[63].2;
ReSlave30.9:=DisplayData[63].3;
ReSlave30.10:=DisplayData[63].4;
ReSlave30.11:=DisplayData[63].5;
ReSlave30.12:=DisplayData[63].6;
ReSlave30.13:=DisplayData[63].7;
ReSlave30.14:=DisplayData[63].9; (*Smoke*)
ReSlave30.15:=DisplayData[63].10; (*Мет*)
(*ReSlave30.14:=DisplayData[51].2;     (*БВВ*)
ReSlave30.15:=DisplayData[51].3;      (*БКДУ*)
ReSlave31.0:=DisplayData[51].4;     (*ЗАШТЫБОВКА*)*)
ReSlave31.1:=DO1;
ReSlave31.2:=Out1.0;
ReSlave31.3:=Out1.1;
ReSlave31.4:=Out1.2;
ReSlave31.5:=Out1.3;
ReSlave31.6:=DI1.1;
ReSlave31.7:=DI1.2;
ReSlave31.8:=In1.3;
ReSlave31.9:=In1.2;
ReSlave31.10:=DisplayData[23].2; (*КТВ*)
ReSlave31.11:=DisplayData[23].3; (*Разгон*)
ReSlave31.12:=DisplayData[23].4;(*Заш*)
ReSlave31.13:=DisplayData[23].5; (*Разрешение*)
ReSlave31.14:=DisplayData[63].10; (*guard*)
ReSlave31.15:=DisplayData[63].11; (*AddAv *)
ReSlave32.0:=In1.6;
ReSlave32.1:=In1.7;
ReSlave32.2:=In1.8;
ReSlave32.3:=In1.9;
(*ReSlave31:=
ReSlave31:=
ReSlave32:=
ReSlave33:=*)


(*
DisplayData[3]:=xDO6Po;
DisplayData[4]:=ZashtibovkaTimePo;
DisplayData[5]:=RazgonTimePo;
DisplayData[6]:=AvariaTimePo;
DisplayData[7]:=PuskTimePo;
DisplayData[8]:=KTBSht;
DisplayData[9]:=TipK1PPo;
DisplayData[10]:=TipK1UPPo;
DisplayData[11]:=TipK2PPo;
DisplayData[12]:=TipK2UPPo;
DisplayData[13]:=TipK3PPo;
DisplayData[14]:=TipK3UPPo;
DisplayData[15]:=TipK4PPo;
DisplayData[16]:=TipK4UPPo;
DisplayData[17]:=NomSpeed;
DisplayData[18]:=DiamKDKS;
DisplayData[19]:=ImpDKS;



xDO6q:=xDO6;
xDO6qi:=xDO6Po;
ZashtibovkaTimeq:=ZashtibovkaTime;
ZashtibovkaTimeqi:=ZashtibovkaTimePo;
RazgonTimeq:=RazgonTime;
RazgonTimeqi:=RazgonTimePo;
AvariaTimeq:=AvariaTime;
AvariaTimeqi:=AvariaTimePo;
PuskTimeq:=PuskTime;
PuskTimeqi:=PuskTimePo;
KTBShtq:=KTBSht;
TipK1q:=TipK1;
TipK1Pq:=TipK1P;
TipK1Pqi:=TipK1PPo;
TipK1Tq:=TipK1T;
TipK1UPq:=TipK1UP;
TipK1UPqi:=TipK1UPPo;
TipK2q:=TipK2;
TipK2Pq:=TipK2P;
TipK2Pqi:=TipK2PPo;
TipK2Tq:=TipK2T;
TipK2UPq:=TipK2UP;
TipK2UPqi:=TipK2UPPo;
TipK3q:=TipK3;
TipK3Pq:=TipK3P;
TipK3Pqi:=TipK3PPo;
TipK3Tq:=TipK3T;
TipK3UPq:=TipK3UP;
TipK3UPqi:=TipK3UPPo;
TipK4q:=TipK4;
TipK4Pq:=TipK4P;
TipK4Pqi:=TipK4PPo;
TipK4Tq:=TipK4T;
TipK4UPq:=TipK4UP;
TipK4UPqi:=TipK4UPPo;
NomSpeedq:=NomSpeed;
TipDatq:=TipDat;
DiamKDKSq:=DiamKDKS;
ImpDKSq:=ImpDKS;
Rezq:=Reztek;





*)
END_PROGRAM
